LIN {X 0,Y 467.337,Z 283.456,A -85,B 0,C 180,E1 -7628.382,E2 -7628.382} C_VEL
LIN {X 0,Y 467.091,Z 291.095,A -85,B 0,C 180,E1 -7631.581,E2 -7631.581} C_VEL
LIN {X 0,Y 466.943,Z 298.315,A -85,B 0,C 180,E1 -7634.545,E2 -7634.545} C_VEL
LIN {X 0,Y 469.161,Z 311.668,A -85,B 0,C 180,E1 -7634.985,E2 -7634.985} C_VEL
LIN {X 0,Y 470.055,Z 319.78,A -85,B 0,C 180,E1 -7635.331,E2 -7635.331} C_VEL
LIN {X 0,Y 469.55,Z 331.872,A -85,B 0,C 180,E1 -7635.924,E2 -7635.924} C_VEL
LIN {X 0,Y 469.022,Z 343.532,A -85,B 0,C 180,E1 -7636.681,E2 -7636.681} C_VEL
LIN {X 0,Y 468.531,Z 353.937,A -85,B 0,C 180,E1 -7637.536,E2 -7637.536} C_VEL
LIN {X 0,Y 468.153,Z 363.71,A -85,B 0,C 180,E1 -7638.527,E2 -7638.527} C_VEL
LIN {X 0,Y 467.611,Z 372.508,A -85,B 0,C 180,E1 -7639.61,E2 -7639.61} C_VEL
LIN {X 0,Y 467.264,Z 381.091,A -85,B 0,C 180,E1 -7640.914,E2 -7640.914} C_VEL
LIN {X 0,Y 466.991,Z 387.971,A -85,B 0,C 180,E1 -7642.216,E2 -7642.216} C_VEL
LIN {X 0,Y 466.835,Z 393.494,A -85,B 0,C 180,E1 -7643.519,E2 -7643.519} C_VEL
LIN {X 0,Y 466.738,Z 397.815,A -85,B 0,C 180,E1 -7644.817,E2 -7644.817} C_VEL
LIN {X 0,Y 466.647,Z 400.107,A -85,B 0,C 180,E1 -7645.682,E2 -7645.682} C_VEL
LIN {X 0,Y 466.689,Z 401.966,A -85,B 0,C 180,E1 -7646.547,E2 -7646.547} C_VEL
LIN {X 0,Y 466.663,Z 403.358,A -85,B 0,C 180,E1 -7647.411,E2 -7647.411} C_VEL
LIN {X 0,Y 466.619,Z 404.96,A -85,B 0,C 180,E1 -7649.137,E2 -7649.137} C_VEL
LIN {X 0,Y 466.599,Z 405.172,A -85,B 0,C 180,E1 -7650,E2 -7650} C_VEL
LIN {X 0,Y 466.619,Z 404.953,A -85,B 0,C 180,E1 -7650.863,E2 -7650.863} C_VEL
LIN {X 0,Y 466.663,Z 403.347,A -85,B 0,C 180,E1 -7652.59,E2 -7652.59} C_VEL
LIN {X 0,Y 466.69,Z 401.945,A -85,B 0,C 180,E1 -7653.453,E2 -7653.453} C_VEL
LIN {X 0,Y 466.69,Z 399,A -85,B 0,C 180,E1 -7654.751,E2 -7654.751} C_VEL
LIN {X 0,Y 466.756,Z 395.011,A -85,B 0,C 180,E1 -7656.05,E2 -7656.05} C_VEL
LIN {X 0,Y 466.951,Z 388.871,A -85,B 0,C 180,E1 -7657.567,E2 -7657.567} C_VEL
LIN {X 0,Y 467.212,Z 382.165,A -85,B 0,C 180,E1 -7658.869,E2 -7658.869} C_VEL
LIN {X 0,Y 467.563,Z 373.843,A -85,B 0,C 180,E1 -7660.172,E2 -7660.172} C_VEL
LIN {X 0,Y 468.003,Z 365.294,A -85,B 0,C 180,E1 -7661.257,E2 -7661.257} C_VEL
LIN {X 0,Y 468.46,Z 355.172,A -85,B 0,C 180,E1 -7662.302,E2 -7662.302} C_VEL
LIN {X 0,Y 468.936,Z 344.257,A -85,B 0,C 180,E1 -7663.212,E2 -7663.212} C_VEL
LIN {X 0,Y 469.451,Z 332.748,A -85,B 0,C 180,E1 -7663.969,E2 -7663.969} C_VEL
LIN {X 0,Y 469.903,Z 320.822,A -85,B 0,C 180,E1 -7664.563,E2 -7664.563} C_VEL
LIN {X 0,Y 469.607,Z 315.894,A -85,B 0,C 180,E1 -7664.774,E2 -7664.774} C_VEL
LIN {X 0,Y 467.679,Z 303.276,A -85,B 0,C 180,E1 -7665.226,E2 -7665.226} C_VEL
LIN {X 0,Y 466.927,Z 298.392,A -85,B 0,C 180,E1 -7665.377,E2 -7665.377} C_VEL
LIN {X 0,Y 467.1,Z 290.512,A -85,B 0,C 180,E1 -7668.575,E2 -7668.575} C_VEL
LIN {X 0,Y 467.335,Z 283.121,A -85,B 0,C 180,E1 -7671.619,E2 -7671.619} C_VEL
LIN {X 0,Y 467.51,Z 275.327,A -85,B 0,C 180,E1 -7674.892,E2 -7674.892} C_VEL
LIN {X 0,Y 467.742,Z 268.646,A -85,B 0,C 180,E1 -7677.76,E2 -7677.76} C_VEL
LIN {X 0,Y 467.985,Z 261.965,A -85,B 0,C 180,E1 -7680.703,E2 -7680.703} C_VEL
LIN {X 0,Y 468.255,Z 256.383,A -85,B 0,C 180,E1 -7683.22,E2 -7683.22} C_VEL
LIN {X 0,Y 468.388,Z 250.837,A -85,B 0,C 180,E1 -7685.815,E2 -7685.815} C_VEL
LIN {X 0,Y 467.612,Z 245.311,A -85,B 0,C 180,E1 -7688.559,E2 -7688.559} C_VEL
LIN {X 0,Y 467.556,Z 245.245,A -85,B 0,C 180,E1 -7691.404,E2 -7691.404} C_VEL
LIN {X 0,Y 467.552,Z 245.247,A -85,B 0,C 180,E1 -7694.948,E2 -7694.948} C_VEL
LIN {X 0,Y 467.554,Z 245.247,A -85,B 0,C 180,E1 -7698.594,E2 -7698.594} C_VEL
LIN {X 0,Y 467.535,Z 245.244,A -85,B 0,C 180,E1 -7701.412,E2 -7701.412} C_VEL
LIN {X 0,Y 467.545,Z 245.247,A -85,B 0,C 180,E1 -7704.262,E2 -7704.262} C_VEL
LIN {X 0,Y 467.575,Z 245.24,A -85,B 0,C 180,E1 -7707.32,E2 -7707.32} C_VEL
LIN {X 0,Y 467.547,Z 245.245,A -85,B 0,C 180,E1 -7710.67,E2 -7710.67} C_VEL
LIN {X 0,Y 467.552,Z 245.243,A -85,B 0,C 180,E1 -7713.195,E2 -7713.195} C_VEL
LIN {X 0,Y 467.583,Z 245.24,A -85,B 0,C 180,E1 -7716.468,E2 -7716.468} C_VEL
LIN {X 0,Y 467.615,Z 245.238,A -85,B 0,C 180,E1 -7719.776,E2 -7719.776} C_VEL
LIN {X 0,Y 467.591,Z 245.239,A -85,B 0,C 180,E1 -7722.505,E2 -7722.505} C_VEL
LIN {X 0,Y 467.598,Z 245.239,A -85,B 0,C 180,E1 -7725.195,E2 -7725.195} C_VEL
LIN {X 0,Y 467.648,Z 245.233,A -85,B 0,C 180,E1 -7727.853,E2 -7727.853} C_VEL
LIN {X 0,Y 467.673,Z 245.231,A -85,B 0,C 180,E1 -7731.356,E2 -7731.356} C_VEL
LIN {X 0,Y 467.734,Z 245.221,A -85,B 0,C 180,E1 -7733.962,E2 -7733.962} C_VEL
LIN {X 0,Y 467.85,Z 245.208,A -85,B 0,C 180,E1 -7737.416,E2 -7737.416} C_VEL
LIN {X 0,Y 467.872,Z 245.204,A -85,B 0,C 180,E1 -7739.999,E2 -7739.999} C_VEL
LIN {X 0,Y 467.851,Z 245.208,A -85,B 0,C 180,E1 -7742.582,E2 -7742.582} C_VEL
LIN {X 0,Y 467.738,Z 245.222,A -85,B 0,C 180,E1 -7746.036,E2 -7746.036} C_VEL
LIN {X 0,Y 467.673,Z 245.23,A -85,B 0,C 180,E1 -7748.642,E2 -7748.642} C_VEL
LIN {X 0,Y 467.646,Z 245.235,A -85,B 0,C 180,E1 -7752.145,E2 -7752.145} C_VEL
LIN {X 0,Y 467.628,Z 245.236,A -85,B 0,C 180,E1 -7755.694,E2 -7755.694} C_VEL
LIN {X 0,Y 467.606,Z 245.237,A -85,B 0,C 180,E1 -7758.764,E2 -7758.764} C_VEL
LIN {X 0,Y 467.569,Z 245.242,A -85,B 0,C 180,E1 -7761.268,E2 -7761.268} C_VEL
LIN {X 0,Y 467.561,Z 245.244,A -85,B 0,C 180,E1 -7763.943,E2 -7763.943} C_VEL
LIN {X 0,Y 467.615,Z 245.235,A -85,B 0,C 180,E1 -7766.799,E2 -7766.799} C_VEL
LIN {X 0,Y 467.575,Z 245.242,A -85,B 0,C 180,E1 -7769.735,E2 -7769.735} C_VEL
LIN {X 0,Y 467.571,Z 245.241,A -85,B 0,C 180,E1 -7772.758,E2 -7772.758} C_VEL
LIN {X 0,Y 467.545,Z 245.243,A -85,B 0,C 180,E1 -7775.889,E2 -7775.889} C_VEL
LIN {X 0,Y 467.606,Z 245.241,A -85,B 0,C 180,E1 -7779.141,E2 -7779.141} C_VEL
LIN {X 0,Y 467.606,Z 245.237,A -85,B 0,C 180,E1 -7782.571,E2 -7782.571} C_VEL
LIN {X 0,Y 467.554,Z 245.241,A -85,B 0,C 180,E1 -7786.177,E2 -7786.177} C_VEL
LIN {X 0,Y 467.569,Z 245.246,A -85,B 0,C 180,E1 -7788.722,E2 -7788.722} C_VEL
LIN {X 0,Y 467.553,Z 245.242,A -85,B 0,C 180,E1 -7791.955,E2 -7791.955} C_VEL
LIN {X 0,Y 467.554,Z 245.242,A -85,B 0,C 180,E1 -7795.167,E2 -7795.167} C_VEL
LIN {X 0,Y 467.57,Z 245.245,A -85,B 0,C 180,E1 -7798.26,E2 -7798.26} C_VEL
LIN {X 0,Y 467.562,Z 245.241,A -85,B 0,C 180,E1 -7801.25,E2 -7801.25} C_VEL
LIN {X 0,Y 467.576,Z 245.245,A -85,B 0,C 180,E1 -7804.159,E2 -7804.159} C_VEL
LIN {X 0,Y 467.497,Z 245.249,A -85,B 0,C 180,E1 -7806.992,E2 -7806.992} C_VEL
LIN {X 0,Y 467.412,Z 245.264,A -85,B 0,C 180,E1 -7807.921,E2 -7807.921} C_VEL
LIN {X 0,Y 467.395,Z 246.234,A -85,B 0,C 180,E1 -7808.846,E2 -7808.846} C_VEL
LIN {X 0,Y 467.382,Z 250.183,A -85,B 0,C 180,E1 -7811.593,E2 -7811.593} C_VEL
LIN {X 0,Y 467.274,Z 254.14,A -85,B 0,C 180,E1 -7814.293,E2 -7814.293} C_VEL
LIN {X 0,Y 467.221,Z 255.612,A -85,B 0,C 180,E1 -7815.284,E2 -7815.284} C_VEL
LIN {X 0,Y 466.522,Z 256.725,A -85,B 0,C 180,E1 -7815.991,E2 -7815.991} C_VEL
LIN {X 0,Y 463.655,Z 258.714,A -85,B 0,C 180,E1 -7817.135,E2 -7817.135} C_VEL
LIN {X 0,Y 461.228,Z 260.326,A -85,B 0,C 180,E1 -7818.057,E2 -7818.057} C_VEL
LIN {X 0,Y 460.157,Z 261.495,A -85,B 0,C 180,E1 -7818.771,E2 -7818.771} C_VEL
LIN {X 0,Y 460.054,Z 261.867,A -85,B 0,C 180,E1 -7819.014,E2 -7819.014} C_VEL
LIN {X 0,Y 459.985,Z 266.526,A -85,B 0,C 180,E1 -7822.096,E2 -7822.096} C_VEL
LIN {X 0,Y 459.995,Z 269.228,A -85,B 0,C 180,E1 -7823.861,E2 -7823.861} C_VEL
LIN {X 0,Y 459.921,Z 273.289,A -85,B 0,C 180,E1 -7826.496,E2 -7826.496} C_VEL
LIN {X 0,Y 459.772,Z 275.027,A -85,B 0,C 180,E1 -7827.509,E2 -7827.509} C_VEL
LIN {X 0,Y 462.387,Z 288.038,A -85,B 0,C 180,E1 -7827.972,E2 -7827.972} C_VEL
LIN {X 0,Y 463.251,Z 293.332,A -85,B 0,C 180,E1 -7828.207,E2 -7828.207} C_VEL
LIN {X 0,Y 462.781,Z 305.595,A -85,B 0,C 180,E1 -7828.803,E2 -7828.803} C_VEL
LIN {X 0,Y 462.304,Z 317.382,A -85,B 0,C 180,E1 -7829.564,E2 -7829.564} C_VEL
LIN {X 0,Y 461.762,Z 329.095,A -85,B 0,C 180,E1 -7830.545,E2 -7830.545} C_VEL
LIN {X 0,Y 461.249,Z 338.561,A -85,B 0,C 180,E1 -7831.528,E2 -7831.528} C_VEL
LIN {X 0,Y 460.775,Z 347.211,A -85,B 0,C 180,E1 -7832.623,E2 -7832.623} C_VEL
LIN {X 0,Y 460.361,Z 355.626,A -85,B 0,C 180,E1 -7833.939,E2 -7833.939} C_VEL
LIN {X 0,Y 459.997,Z 362.401,A -85,B 0,C 180,E1 -7835.26,E2 -7835.26} C_VEL
LIN {X 0,Y 459.885,Z 367.999,A -85,B 0,C 180,E1 -7836.633,E2 -7836.633} C_VEL
LIN {X 0,Y 459.742,Z 372.063,A -85,B 0,C 180,E1 -7837.908,E2 -7837.908} C_VEL
LIN {X 0,Y 459.618,Z 374.329,A -85,B 0,C 180,E1 -7838.795,E2 -7838.795} C_VEL
LIN {X 0,Y 459.525,Z 376.121,A -85,B 0,C 180,E1 -7839.685,E2 -7839.685} C_VEL
LIN {X 0,Y 459.538,Z 377.468,A -85,B 0,C 180,E1 -7840.575,E2 -7840.575} C_VEL
LIN {X 0,Y 459.549,Z 378.692,A -85,B 0,C 180,E1 -7841.836,E2 -7841.836} C_VEL
LIN {X 0,Y 459.433,Z 379.083,A -85,B 0,C 180,E1 -7843.265,E2 -7843.265} C_VEL
LIN {X 0,Y 459.442,Z 378.784,A -85,B 0,C 180,E1 -7844.167,E2 -7844.167} C_VEL
LIN {X 0,Y 459.507,Z 377.557,A -85,B 0,C 180,E1 -7845.521,E2 -7845.521} C_VEL
LIN {X 0,Y 459.619,Z 374.388,A -85,B 0,C 180,E1 -7847.347,E2 -7847.347} C_VEL
LIN {X 0,Y 459.789,Z 370.739,A -85,B 0,C 180,E1 -7848.722,E2 -7848.722} C_VEL
LIN {X 0,Y 459.959,Z 365.869,A -85,B 0,C 180,E1 -7850.108,E2 -7850.108} C_VEL
LIN {X 0,Y 460.265,Z 359.619,A -85,B 0,C 180,E1 -7851.497,E2 -7851.497} C_VEL
LIN {X 0,Y 460.667,Z 351.74,A -85,B 0,C 180,E1 -7852.894,E2 -7852.894} C_VEL
LIN {X 0,Y 461.173,Z 342.78,A -85,B 0,C 180,E1 -7854.156,E2 -7854.156} C_VEL
LIN {X 0,Y 461.731,Z 332.286,A -85,B 0,C 180,E1 -7855.346,E2 -7855.346} C_VEL
LIN {X 0,Y 462.268,Z 321.584,A -85,B 0,C 180,E1 -7856.315,E2 -7856.315} C_VEL
LIN {X 0,Y 462.77,Z 310.611,A -85,B 0,C 180,E1 -7857.103,E2 -7857.103} C_VEL
LIN {X 0,Y 463.317,Z 299.025,A -85,B 0,C 180,E1 -7857.747,E2 -7857.747} C_VEL
LIN {X 0,Y 463.379,Z 292.5,A -85,B 0,C 180,E1 -7858.045,E2 -7858.045} C_VEL
LIN {X 0,Y 460.857,Z 279.894,A -85,B 0,C 180,E1 -7858.577,E2 -7858.577} C_VEL
LIN {X 0,Y 459.719,Z 275.001,A -85,B 0,C 180,E1 -7858.759,E2 -7858.759} C_VEL
LIN {X 0,Y 459.8,Z 271.128,A -85,B 0,C 180,E1 -7861.31,E2 -7861.31} C_VEL
LIN {X 0,Y 459.943,Z 266.479,A -85,B 0,C 180,E1 -7864.427,E2 -7864.427} C_VEL
LIN {X 0,Y 460.058,Z 261.784,A -85,B 0,C 180,E1 -7867.665,E2 -7867.665} C_VEL
LIN {X 0,Y 460.159,Z 258.147,A -85,B 0,C 180,E1 -7870.215,E2 -7870.215} C_VEL
LIN {X 0,Y 460.334,Z 253.735,A -85,B 0,C 180,E1 -7873.394,E2 -7873.394} C_VEL
LIN {X 0,Y 460.478,Z 250.436,A -85,B 0,C 180,E1 -7875.833,E2 -7875.833} C_VEL
LIN {X 0,Y 460.5,Z 247.076,A -85,B 0,C 180,E1 -7878.4,E2 -7878.4} C_VEL
LIN {X 0,Y 460.468,Z 246.334,A -85,B 0,C 180,E1 -7878.984,E2 -7878.984} C_VEL
LIN {X 0,Y 460.503,Z 246.128,A -85,B 0,C 180,E1 -7881.266,E2 -7881.266} C_VEL
LIN {X 0,Y 460.5,Z 246.126,A -85,B 0,C 180,E1 -7884.555,E2 -7884.555} C_VEL
LIN {X 0,Y 460.519,Z 246.123,A -85,B 0,C 180,E1 -7887.716,E2 -7887.716} C_VEL
LIN {X 0,Y 460.534,Z 246.119,A -85,B 0,C 180,E1 -7890.77,E2 -7890.77} C_VEL
LIN {X 0,Y 460.55,Z 246.118,A -85,B 0,C 180,E1 -7893.735,E2 -7893.735} C_VEL
LIN {X 0,Y 460.539,Z 246.118,A -85,B 0,C 180,E1 -7896.625,E2 -7896.625} C_VEL
LIN {X 0,Y 460.561,Z 246.117,A -85,B 0,C 180,E1 -7899.455,E2 -7899.455} C_VEL
LIN {X 0,Y 460.547,Z 246.118,A -85,B 0,C 180,E1 -7902.231,E2 -7902.231} C_VEL
LIN {X 0,Y 460.556,Z 246.116,A -85,B 0,C 180,E1 -7904.966,E2 -7904.966} C_VEL
LIN {X 0,Y 460.6,Z 246.113,A -85,B 0,C 180,E1 -7908.56,E2 -7908.56} C_VEL
LIN {X 0,Y 460.684,Z 246.099,A -85,B 0,C 180,E1 -7912.109,E2 -7912.109} C_VEL
LIN {X 0,Y 460.681,Z 246.102,A -85,B 0,C 180,E1 -7914.749,E2 -7914.749} C_VEL
LIN {X 0,Y 460.816,Z 246.087,A -85,B 0,C 180,E1 -7917.379,E2 -7917.379} C_VEL
LIN {X 0,Y 460.839,Z 246.08,A -85,B 0,C 180,E1 -7920.001,E2 -7920.001} C_VEL
LIN {X 0,Y 460.817,Z 246.083,A -85,B 0,C 180,E1 -7922.623,E2 -7922.623} C_VEL
LIN {X 0,Y 460.691,Z 246.099,A -85,B 0,C 180,E1 -7926.131,E2 -7926.131} C_VEL
LIN {X 0,Y 460.62,Z 246.108,A -85,B 0,C 180,E1 -7928.777,E2 -7928.777} C_VEL
LIN {X 0,Y 460.605,Z 246.113,A -85,B 0,C 180,E1 -7932.446,E2 -7932.446} C_VEL
LIN {X 0,Y 460.593,Z 246.114,A -85,B 0,C 180,E1 -7935.999,E2 -7935.999} C_VEL
LIN {X 0,Y 460.563,Z 246.118,A -85,B 0,C 180,E1 -7938.903,E2 -7938.903} C_VEL
LIN {X 0,Y 460.509,Z 246.126,A -85,B 0,C 180,E1 -7941.487,E2 -7941.487} C_VEL
LIN {X 0,Y 460.534,Z 246.123,A -85,B 0,C 180,E1 -7944.334,E2 -7944.334} C_VEL
LIN {X 0,Y 460.531,Z 246.123,A -85,B 0,C 180,E1 -7947.247,E2 -7947.247} C_VEL
LIN {X 0,Y 460.503,Z 246.125,A -85,B 0,C 180,E1 -7950.241,E2 -7950.241} C_VEL
LIN {X 0,Y 460.525,Z 246.122,A -85,B 0,C 180,E1 -7953.326,E2 -7953.326} C_VEL
LIN {X 0,Y 460.472,Z 246.129,A -85,B 0,C 180,E1 -7956.531,E2 -7956.531} C_VEL
LIN {X 0,Y 460.529,Z 246.119,A -85,B 0,C 180,E1 -7959.864,E2 -7959.864} C_VEL
LIN {X 0,Y 460.511,Z 246.124,A -85,B 0,C 180,E1 -7962.902,E2 -7962.902} C_VEL
LIN {X 0,Y 460.501,Z 246.126,A -85,B 0,C 180,E1 -7965.833,E2 -7965.833} C_VEL
LIN {X 0,Y 460.515,Z 246.126,A -85,B 0,C 180,E1 -7968.988,E2 -7968.988} C_VEL
LIN {X 0,Y 460.544,Z 246.294,A -85,B 0,C 180,E1 -7970.039,E2 -7970.039} C_VEL
LIN {X 0,Y 461.414,Z 251.524,A -85,B 0,C 180,E1 -7973.014,E2 -7973.014} C_VEL
LIN {X 0,Y 461.641,Z 255.871,A -85,B 0,C 180,E1 -7975.296,E2 -7975.296} C_VEL
LIN {X 0,Y 461.246,Z 262.522,A -85,B 0,C 180,E1 -7978.57,E2 -7978.57} C_VEL
LIN {X 0,Y 460.92,Z 268.312,A -85,B 0,C 180,E1 -7981.295,E2 -7981.295} C_VEL
LIN {X 0,Y 460.542,Z 275.812,A -85,B 0,C 180,E1 -7984.705,E2 -7984.705} C_VEL
LIN {X 0,Y 460.29,Z 283.369,A -85,B 0,C 180,E1 -7988.033,E2 -7988.033} C_VEL
LIN {X 0,Y 460.019,Z 291.021,A -85,B 0,C 180,E1 -7991.302,E2 -7991.302} C_VEL
LIN {X 0,Y 459.866,Z 298.093,A -85,B 0,C 180,E1 -7994.271,E2 -7994.271} C_VEL
LIN {X 0,Y 462.203,Z 311.72,A -85,B 0,C 180,E1 -7994.741,E2 -7994.741} C_VEL
LIN {X 0,Y 463.181,Z 320.041,A -85,B 0,C 180,E1 -7995.108,E2 -7995.108} C_VEL
LIN {X 0,Y 462.671,Z 332.016,A -85,B 0,C 180,E1 -7995.71,E2 -7995.71} C_VEL
LIN {X 0,Y 462.121,Z 343.569,A -85,B 0,C 180,E1 -7996.478,E2 -7996.478} C_VEL
LIN {X 0,Y 461.565,Z 354.304,A -85,B 0,C 180,E1 -7997.381,E2 -7997.381} C_VEL
LIN {X 0,Y 461.173,Z 363.657,A -85,B 0,C 180,E1 -7998.351,E2 -7998.351} C_VEL
LIN {X 0,Y 460.602,Z 372.425,A -85,B 0,C 180,E1 -7999.45,E2 -7999.45} C_VEL
LIN {X 0,Y 460.231,Z 380.975,A -85,B 0,C 180,E1 -8000.774,E2 -8000.774} C_VEL
LIN {X 0,Y 459.93,Z 387.835,A -85,B 0,C 180,E1 -8002.096,E2 -8002.096} C_VEL
LIN {X 0,Y 459.744,Z 393.784,A -85,B 0,C 180,E1 -8003.539,E2 -8003.539} C_VEL
LIN {X 0,Y 459.618,Z 398.866,A -85,B 0,C 180,E1 -8005.176,E2 -8005.176} C_VEL
LIN {X 0,Y 459.584,Z 401.786,A -85,B 0,C 180,E1 -8006.493,E2 -8006.493} C_VEL
LIN {X 0,Y 459.585,Z 403.173,A -85,B 0,C 180,E1 -8007.371,E2 -8007.371} C_VEL
LIN {X 0,Y 459.522,Z 404.766,A -85,B 0,C 180,E1 -8009.124,E2 -8009.124} C_VEL
LIN {X 0,Y 459.53,Z 404.972,A -85,B 0,C 180,E1 -8010,E2 -8010} C_VEL
LIN {X 0,Y 459.521,Z 404.133,A -85,B 0,C 180,E1 -8011.753,E2 -8011.753} C_VEL
LIN {X 0,Y 459.585,Z 403.133,A -85,B 0,C 180,E1 -8012.629,E2 -8012.629} C_VEL
LIN {X 0,Y 459.585,Z 401.722,A -85,B 0,C 180,E1 -8013.507,E2 -8013.507} C_VEL
LIN {X 0,Y 459.618,Z 398.769,A -85,B 0,C 180,E1 -8014.824,E2 -8014.824} C_VEL
LIN {X 0,Y 459.716,Z 393.725,A -85,B 0,C 180,E1 -8016.431,E2 -8016.431} C_VEL
LIN {X 0,Y 459.911,Z 387.593,A -85,B 0,C 180,E1 -8017.905,E2 -8017.905} C_VEL
LIN {X 0,Y 460.231,Z 380.642,A -85,B 0,C 180,E1 -8019.227,E2 -8019.227} C_VEL
LIN {X 0,Y 460.594,Z 371.921,A -85,B 0,C 180,E1 -8020.55,E2 -8020.55} C_VEL
LIN {X 0,Y 461.092,Z 362.99,A -85,B 0,C 180,E1 -8021.651,E2 -8021.651} C_VEL
LIN {X 0,Y 461.59,Z 352.085,A -85,B 0,C 180,E1 -8022.743,E2 -8022.743} C_VEL
LIN {X 0,Y 462.117,Z 340.786,A -85,B 0,C 180,E1 -8023.634,E2 -8023.634} C_VEL
LIN {X 0,Y 462.693,Z 328.254,A -85,B 0,C 180,E1 -8024.402,E2 -8024.402} C_VEL
LIN {X 0,Y 462.962,Z 318.886,A -85,B 0,C 180,E1 -8024.843,E2 -8024.843} C_VEL
LIN {X 0,Y 461.078,Z 305.955,A -85,B 0,C 180,E1 -8025.356,E2 -8025.356} C_VEL
LIN {X 0,Y 459.847,Z 298.205,A -85,B 0,C 180,E1 -8025.599,E2 -8025.599} C_VEL
LIN {X 0,Y 460.07,Z 289.556,A -85,B 0,C 180,E1 -8029.173,E2 -8029.173} C_VEL
LIN {X 0,Y 460.281,Z 281.788,A -85,B 0,C 180,E1 -8032.44,E2 -8032.44} C_VEL
LIN {X 0,Y 460.561,Z 273.953,A -85,B 0,C 180,E1 -8035.799,E2 -8035.799} C_VEL
LIN {X 0,Y 460.826,Z 266.206,A -85,B 0,C 180,E1 -8039.21,E2 -8039.21} C_VEL
LIN {X 0,Y 461.165,Z 259.53,A -85,B 0,C 180,E1 -8042.234,E2 -8042.234} C_VEL
LIN {X 0,Y 461.405,Z 252.861,A -85,B 0,C 180,E1 -8045.366,E2 -8045.366} C_VEL
LIN {X 0,Y 460.917,Z 248.389,A -85,B 0,C 180,E1 -8047.582,E2 -8047.582} C_VEL
LIN {X 0,Y 460.555,Z 246.12,A -85,B 0,C 180,E1 -8048.822,E2 -8048.822} C_VEL
LIN {X 0,Y 460.471,Z 246.126,A -85,B 0,C 180,E1 -8052.186,E2 -8052.186} C_VEL
LIN {X 0,Y 460.494,Z 246.122,A -85,B 0,C 180,E1 -8055.408,E2 -8055.408} C_VEL
LIN {X 0,Y 460.51,Z 246.122,A -85,B 0,C 180,E1 -8058.986,E2 -8058.986} C_VEL
LIN {X 0,Y 460.477,Z 246.127,A -85,B 0,C 180,E1 -8062.374,E2 -8062.374} C_VEL
LIN {X 0,Y 460.529,Z 246.118,A -85,B 0,C 180,E1 -8065.621,E2 -8065.621} C_VEL
LIN {X 0,Y 460.533,Z 246.118,A -85,B 0,C 180,E1 -8068.743,E2 -8068.743} C_VEL
LIN {X 0,Y 460.534,Z 246.122,A -85,B 0,C 180,E1 -8072.263,E2 -8072.263} C_VEL
LIN {X 0,Y 460.528,Z 246.118,A -85,B 0,C 180,E1 -8074.703,E2 -8074.703} C_VEL
LIN {X 0,Y 460.504,Z 246.123,A -85,B 0,C 180,E1 -8077.57,E2 -8077.57} C_VEL
LIN {X 0,Y 460.561,Z 246.115,A -85,B 0,C 180,E1 -8080.383,E2 -8080.383} C_VEL
LIN {X 0,Y 460.597,Z 246.111,A -85,B 0,C 180,E1 -8084.058,E2 -8084.058} C_VEL
LIN {X 0,Y 460.601,Z 246.113,A -85,B 0,C 180,E1 -8087.665,E2 -8087.665} C_VEL
LIN {X 0,Y 460.62,Z 246.109,A -85,B 0,C 180,E1 -8091.223,E2 -8091.223} C_VEL
LIN {X 0,Y 460.7,Z 246.098,A -85,B 0,C 180,E1 -8093.869,E2 -8093.869} C_VEL
LIN {X 0,Y 460.815,Z 246.085,A -85,B 0,C 180,E1 -8097.377,E2 -8097.377} C_VEL
LIN {X 0,Y 460.843,Z 246.08,A -85,B 0,C 180,E1 -8099.999,E2 -8099.999} C_VEL
LIN {X 0,Y 460.816,Z 246.084,A -85,B 0,C 180,E1 -8102.621,E2 -8102.621} C_VEL
LIN {X 0,Y 460.703,Z 246.1,A -85,B 0,C 180,E1 -8106.129,E2 -8106.129} C_VEL
LIN {X 0,Y 460.62,Z 246.108,A -85,B 0,C 180,E1 -8108.775,E2 -8108.775} C_VEL
LIN {X 0,Y 460.602,Z 246.11,A -85,B 0,C 180,E1 -8112.444,E2 -8112.444} C_VEL
LIN {X 0,Y 460.589,Z 246.114,A -85,B 0,C 180,E1 -8115.997,E2 -8115.997} C_VEL
LIN {X 0,Y 460.559,Z 246.114,A -85,B 0,C 180,E1 -8118.901,E2 -8118.901} C_VEL
LIN {X 0,Y 460.504,Z 246.124,A -85,B 0,C 180,E1 -8121.485,E2 -8121.485} C_VEL
LIN {X 0,Y 460.53,Z 246.118,A -85,B 0,C 180,E1 -8124.332,E2 -8124.332} C_VEL
LIN {X 0,Y 460.572,Z 246.115,A -85,B 0,C 180,E1 -8127.242,E2 -8127.242} C_VEL
LIN {X 0,Y 460.515,Z 246.119,A -85,B 0,C 180,E1 -8130.238,E2 -8130.238} C_VEL
LIN {X 0,Y 460.517,Z 246.124,A -85,B 0,C 180,E1 -8133.324,E2 -8133.324} C_VEL
LIN {X 0,Y 460.468,Z 246.125,A -85,B 0,C 180,E1 -8136.528,E2 -8136.528} C_VEL
LIN {X 0,Y 460.566,Z 246.112,A -85,B 0,C 180,E1 -8139.857,E2 -8139.857} C_VEL
LIN {X 0,Y 460.53,Z 246.123,A -85,B 0,C 180,E1 -8142.904,E2 -8142.904} C_VEL
LIN {X 0,Y 460.506,Z 246.118,A -85,B 0,C 180,E1 -8145.829,E2 -8145.829} C_VEL
LIN {X 0,Y 460.521,Z 246.121,A -85,B 0,C 180,E1 -8148.989,E2 -8148.989} C_VEL
LIN {X 0,Y 460.513,Z 246.119,A -85,B 0,C 180,E1 -8151.267,E2 -8151.267} C_VEL
LIN {X 0,Y 460.5,Z 246.126,A -85,B 0,C 180,E1 -8154.554,E2 -8154.554} C_VEL
LIN {X 0,Y 460.519,Z 246.119,A -85,B 0,C 180,E1 -8157.715,E2 -8157.715} C_VEL
LIN {X 0,Y 460.526,Z 246.119,A -85,B 0,C 180,E1 -8160.769,E2 -8160.769} C_VEL
LIN {X 0,Y 460.53,Z 246.119,A -85,B 0,C 180,E1 -8163.733,E2 -8163.733} C_VEL
LIN {X 0,Y 460.493,Z 246.123,A -85,B 0,C 180,E1 -8166.622,E2 -8166.622} C_VEL
LIN {X 0,Y 460.394,Z 246.136,A -85,B 0,C 180,E1 -8167.566,E2 -8167.566} C_VEL
LIN {X 0,Y 460.351,Z 246.764,A -85,B 0,C 180,E1 -8168.628,E2 -8168.628} C_VEL
LIN {X 0,Y 460.336,Z 250.56,A -85,B 0,C 180,E1 -8171.301,E2 -8171.301} C_VEL
LIN {X 0,Y 460.208,Z 254.705,A -85,B 0,C 180,E1 -8174.168,E2 -8174.168} C_VEL
LIN {X 0,Y 460.179,Z 260.044,A -85,B 0,C 180,E1 -8177.796,E2 -8177.796} C_VEL
LIN {X 0,Y 460.054,Z 261.867,A -85,B 0,C 180,E1 -8179.014,E2 -8179.014} C_VEL
LIN {X 0,Y 459.332,Z 263.009,A -85,B 0,C 180,E1 -8179.73,E2 -8179.73} C_VEL
LIN {X 0,Y 456.425,Z 265.021,A -85,B 0,C 180,E1 -8180.889,E2 -8180.889} C_VEL
LIN {X 0,Y 454.015,Z 266.644,A -85,B 0,C 180,E1 -8181.824,E2 -8181.824} C_VEL
LIN {X 0,Y 453.012,Z 267.825,A -85,B 0,C 180,E1 -8182.548,E2 -8182.548} C_VEL
LIN {X 0,Y 452.946,Z 268.201,A -85,B 0,C 180,E1 -8182.793,E2 -8182.793} C_VEL
LIN {X 0,Y 452.9,Z 272.381,A -85,B 0,C 180,E1 -8185.55,E2 -8185.55} C_VEL
LIN {X 0,Y 452.753,Z 275.057,A -85,B 0,C 180,E1 -8187.275,E2 -8187.275} C_VEL
LIN {X 0,Y 455.252,Z 288.015,A -85,B 0,C 180,E1 -8187.747,E2 -8187.747} C_VEL
LIN {X 0,Y 456.35,Z 293.838,A -85,B 0,C 180,E1 -8188.014,E2 -8188.014} C_VEL
LIN {X 0,Y 455.884,Z 305.059,A -85,B 0,C 180,E1 -8188.565,E2 -8188.565} C_VEL
LIN {X 0,Y 455.405,Z 317.014,A -85,B 0,C 180,E1 -8189.337,E2 -8189.337} C_VEL
LIN {X 0,Y 454.855,Z 327.71,A -85,B 0,C 180,E1 -8190.221,E2 -8190.221} C_VEL
LIN {X 0,Y 454.265,Z 338.411,A -85,B 0,C 180,E1 -8191.33,E2 -8191.33} C_VEL
LIN {X 0,Y 453.783,Z 347.119,A -85,B 0,C 180,E1 -8192.441,E2 -8192.441} C_VEL
LIN {X 0,Y 453.316,Z 355.609,A -85,B 0,C 180,E1 -8193.778,E2 -8193.778} C_VEL
LIN {X 0,Y 452.944,Z 362.424,A -85,B 0,C 180,E1 -8195.118,E2 -8195.118} C_VEL
LIN {X 0,Y 452.804,Z 368.465,A -85,B 0,C 180,E1 -8196.626,E2 -8196.626} C_VEL
LIN {X 0,Y 452.647,Z 372.78,A -85,B 0,C 180,E1 -8198.032,E2 -8198.032} C_VEL
LIN {X 0,Y 452.51,Z 374.934,A -85,B 0,C 180,E1 -8198.935,E2 -8198.935} C_VEL
LIN {X 0,Y 452.429,Z 376.625,A -85,B 0,C 180,E1 -8199.838,E2 -8199.838} C_VEL
LIN {X 0,Y 452.437,Z 377.905,A -85,B 0,C 180,E1 -8200.743,E2 -8200.743} C_VEL
LIN {X 0,Y 452.447,Z 378.918,A -85,B 0,C 180,E1 -8201.883,E2 -8201.883} C_VEL
LIN {X 0,Y 452.345,Z 379.25,A -85,B 0,C 180,E1 -8203.476,E2 -8203.476} C_VEL
LIN {X 0,Y 452.354,Z 378.883,A -85,B 0,C 180,E1 -8204.393,E2 -8204.393} C_VEL
LIN {X 0,Y 452.427,Z 377.709,A -85,B 0,C 180,E1 -8205.618,E2 -8205.618} C_VEL
LIN {X 0,Y 452.496,Z 375.156,A -85,B 0,C 180,E1 -8207.163,E2 -8207.163} C_VEL
LIN {X 0,Y 452.707,Z 371.21,A -85,B 0,C 180,E1 -8208.745,E2 -8208.745} C_VEL
LIN {X 0,Y 452.864,Z 367.133,A -85,B 0,C 180,E1 -8209.963,E2 -8209.963} C_VEL
LIN {X 0,Y 453.203,Z 360.564,A -85,B 0,C 180,E1 -8211.5,E2 -8211.5} C_VEL
LIN {X 0,Y 453.593,Z 353.619,A -85,B 0,C 180,E1 -8212.789,E2 -8212.789} C_VEL
LIN {X 0,Y 454.092,Z 345.186,A -85,B 0,C 180,E1 -8214.06,E2 -8214.06} C_VEL
LIN {X 0,Y 454.618,Z 336.264,A -85,B 0,C 180,E1 -8215.158,E2 -8215.158} C_VEL
LIN {X 0,Y 455.213,Z 325.906,A -85,B 0,C 180,E1 -8216.188,E2 -8216.188} C_VEL
LIN {X 0,Y 455.762,Z 314.997,A -85,B 0,C 180,E1 -8217.058,E2 -8217.058} C_VEL
LIN {X 0,Y 456.342,Z 303.508,A -85,B 0,C 180,E1 -8217.776,E2 -8217.776} C_VEL
LIN {X 0,Y 456.504,Z 293.308,A -85,B 0,C 180,E1 -8218.275,E2 -8218.275} C_VEL
LIN {X 0,Y 454.092,Z 281.17,A -85,B 0,C 180,E1 -8218.812,E2 -8218.812} C_VEL
LIN {X 0,Y 452.648,Z 275.183,A -85,B 0,C 180,E1 -8219.057,E2 -8219.057} C_VEL
LIN {X 0,Y 452.738,Z 270.993,A -85,B 0,C 180,E1 -8221.856,E2 -8221.856} C_VEL
LIN {X 0,Y 452.877,Z 266.334,A -85,B 0,C 180,E1 -8225.042,E2 -8225.042} C_VEL
LIN {X 0,Y 453.033,Z 261.603,A -85,B 0,C 180,E1 -8228.354,E2 -8228.354} C_VEL
LIN {X 0,Y 453.154,Z 256.782,A -85,B 0,C 180,E1 -8231.826,E2 -8231.826} C_VEL
LIN {X 0,Y 453.373,Z 253.147,A -85,B 0,C 180,E1 -8234.517,E2 -8234.517} C_VEL
LIN {X 0,Y 453.468,Z 249.862,A -85,B 0,C 180,E1 -8237.008,E2 -8237.008} C_VEL
LIN {X 0,Y 453.453,Z 247.009,A -85,B 0,C 180,E1 -8239.414,E2 -8239.414} C_VEL
LIN {X 0,Y 453.458,Z 247.003,A -85,B 0,C 180,E1 -8242.813,E2 -8242.813} C_VEL
LIN {X 0,Y 453.465,Z 247.004,A -85,B 0,C 180,E1 -8246.088,E2 -8246.088} C_VEL
LIN {X 0,Y 453.47,Z 247,A -85,B 0,C 180,E1 -8249.242,E2 -8249.242} C_VEL
LIN {X 0,Y 453.524,Z 246.992,A -85,B 0,C 180,E1 -8252.298,E2 -8252.298} C_VEL
LIN {X 0,Y 453.503,Z 246.995,A -85,B 0,C 180,E1 -8255.266,E2 -8255.266} C_VEL
LIN {X 0,Y 453.524,Z 246.992,A -85,B 0,C 180,E1 -8258.398,E2 -8258.398} C_VEL
LIN {X 0,Y 453.51,Z 246.996,A -85,B 0,C 180,E1 -8261.009,E2 -8261.009} C_VEL
LIN {X 0,Y 453.564,Z 246.991,A -85,B 0,C 180,E1 -8263.877,E2 -8263.877} C_VEL
LIN {X 0,Y 453.552,Z 246.988,A -85,B 0,C 180,E1 -8267.472,E2 -8267.472} C_VEL
LIN {X 0,Y 453.582,Z 246.986,A -85,B 0,C 180,E1 -8271.088,E2 -8271.088} C_VEL
LIN {X 0,Y 453.655,Z 246.974,A -85,B 0,C 180,E1 -8273.776,E2 -8273.776} C_VEL
LIN {X 0,Y 453.757,Z 246.966,A -85,B 0,C 180,E1 -8277.338,E2 -8277.338} C_VEL
LIN {X 0,Y 453.81,Z 246.955,A -85,B 0,C 180,E1 -8280.001,E2 -8280.001} C_VEL
LIN {X 0,Y 453.757,Z 246.963,A -85,B 0,C 180,E1 -8282.664,E2 -8282.664} C_VEL
LIN {X 0,Y 453.659,Z 246.975,A -85,B 0,C 180,E1 -8286.227,E2 -8286.227} C_VEL
LIN {X 0,Y 453.584,Z 246.984,A -85,B 0,C 180,E1 -8288.915,E2 -8288.915} C_VEL
LIN {X 0,Y 453.556,Z 246.992,A -85,B 0,C 180,E1 -8292.53,E2 -8292.53} C_VEL
LIN {X 0,Y 453.537,Z 246.992,A -85,B 0,C 180,E1 -8296.197,E2 -8296.197} C_VEL
LIN {X 0,Y 453.513,Z 246.996,A -85,B 0,C 180,E1 -8299.042,E2 -8299.042} C_VEL
LIN {X 0,Y 453.47,Z 247.003,A -85,B 0,C 180,E1 -8301.837,E2 -8301.837} C_VEL
LIN {X 0,Y 453.503,Z 247.001,A -85,B 0,C 180,E1 -8304.736,E2 -8304.736} C_VEL
LIN {X 0,Y 453.5,Z 246.999,A -85,B 0,C 180,E1 -8307.954,E2 -8307.954} C_VEL
LIN {X 0,Y 453.47,Z 247.003,A -85,B 0,C 180,E1 -8310.761,E2 -8310.761} C_VEL
LIN {X 0,Y 453.472,Z 247.001,A -85,B 0,C 180,E1 -8313.914,E2 -8313.914} C_VEL
LIN {X 0,Y 453.448,Z 247.002,A -85,B 0,C 180,E1 -8317.191,E2 -8317.191} C_VEL
LIN {X 0,Y 453.502,Z 246.996,A -85,B 0,C 180,E1 -8319.449,E2 -8319.449} C_VEL
LIN {X 0,Y 453.461,Z 247.003,A -85,B 0,C 180,E1 -8322.996,E2 -8322.996} C_VEL
LIN {X 0,Y 453.456,Z 247.002,A -85,B 0,C 180,E1 -8325.779,E2 -8325.779} C_VEL
LIN {X 0,Y 453.496,Z 246.999,A -85,B 0,C 180,E1 -8329.596,E2 -8329.596} C_VEL
LIN {X 0,Y 454.425,Z 252.628,A -85,B 0,C 180,E1 -8332.904,E2 -8332.904} C_VEL
LIN {X 0,Y 454.638,Z 256.744,A -85,B 0,C 180,E1 -8335.114,E2 -8335.114} C_VEL
LIN {X 0,Y 454.328,Z 261.957,A -85,B 0,C 180,E1 -8337.746,E2 -8337.746} C_VEL
LIN {X 0,Y 453.961,Z 268.284,A -85,B 0,C 180,E1 -8340.813,E2 -8340.813} C_VEL
LIN {X 0,Y 453.533,Z 275.748,A -85,B 0,C 180,E1 -8344.286,E2 -8344.286} C_VEL
LIN {X 0,Y 453.251,Z 283.29,A -85,B 0,C 180,E1 -8347.674,E2 -8347.674} C_VEL
LIN {X 0,Y 453.041,Z 289.788,A -85,B 0,C 180,E1 -8350.517,E2 -8350.517} C_VEL
LIN {X 0,Y 452.832,Z 297.904,A -85,B 0,C 180,E1 -8353.997,E2 -8353.997} C_VEL
LIN {X 0,Y 455.216,Z 311.642,A -85,B 0,C 180,E1 -8354.48,E2 -8354.48} C_VEL
LIN {X 0,Y 456.324,Z 321.665,A -85,B 0,C 180,E1 -8354.936,E2 -8354.936} C_VEL
LIN {X 0,Y 455.713,Z 333.987,A -85,B 0,C 180,E1 -8355.601,E2 -8355.601} C_VEL
LIN {X 0,Y 455.048,Z 346.499,A -85,B 0,C 180,E1 -8356.491,E2 -8356.491} C_VEL
LIN {X 0,Y 454.553,Z 356.142,A -85,B 0,C 180,E1 -8357.359,E2 -8357.359} C_VEL
LIN {X 0,Y 454.113,Z 365.546,A -85,B 0,C 180,E1 -8358.394,E2 -8358.394} C_VEL
LIN {X 0,Y 453.509,Z 373.915,A -85,B 0,C 180,E1 -8359.509,E2 -8359.509} C_VEL
LIN {X 0,Y 453.117,Z 382.114,A -85,B 0,C 180,E1 -8360.853,E2 -8360.853} C_VEL
LIN {X 0,Y 452.865,Z 387.717,A -85,B 0,C 180,E1 -8361.971,E2 -8361.971} C_VEL
LIN {X 0,Y 452.653,Z 394.09,A -85,B 0,C 180,E1 -8363.56,E2 -8363.56} C_VEL
LIN {X 0,Y 452.546,Z 398.706,A -85,B 0,C 180,E1 -8365.1,E2 -8365.1} C_VEL
LIN {X 0,Y 452.48,Z 401.613,A -85,B 0,C 180,E1 -8366.438,E2 -8366.438} C_VEL
LIN {X 0,Y 452.509,Z 402.993,A -85,B 0,C 180,E1 -8367.33,E2 -8367.33} C_VEL
LIN {X 0,Y 452.429,Z 404.574,A -85,B 0,C 180,E1 -8369.11,E2 -8369.11} C_VEL
LIN {X 0,Y 452.435,Z 404.771,A -85,B 0,C 180,E1 -8370,E2 -8370} C_VEL
LIN {X 0,Y 452.437,Z 403.919,A -85,B 0,C 180,E1 -8371.78,E2 -8371.78} C_VEL
LIN {X 0,Y 452.509,Z 402.913,A -85,B 0,C 180,E1 -8372.671,E2 -8372.671} C_VEL
LIN {X 0,Y 452.481,Z 401.491,A -85,B 0,C 180,E1 -8373.562,E2 -8373.562} C_VEL
LIN {X 0,Y 452.546,Z 398.527,A -85,B 0,C 180,E1 -8374.9,E2 -8374.9} C_VEL
LIN {X 0,Y 452.613,Z 393.956,A -85,B 0,C 180,E1 -8376.396,E2 -8376.396} C_VEL
LIN {X 0,Y 452.857,Z 387.312,A -85,B 0,C 180,E1 -8378.029,E2 -8378.029} C_VEL
LIN {X 0,Y 453.2,Z 380.335,A -85,B 0,C 180,E1 -8379.371,E2 -8379.371} C_VEL
LIN {X 0,Y 453.572,Z 371.578,A -85,B 0,C 180,E1 -8380.716,E2 -8380.716} C_VEL
LIN {X 0,Y 454.103,Z 362.613,A -85,B 0,C 180,E1 -8381.833,E2 -8381.833} C_VEL
LIN {X 0,Y 454.602,Z 352.363,A -85,B 0,C 180,E1 -8382.877,E2 -8382.877} C_VEL
LIN {X 0,Y 455.098,Z 341.877,A -85,B 0,C 180,E1 -8383.735,E2 -8383.735} C_VEL
LIN {X 0,Y 455.685,Z 329.667,A -85,B 0,C 180,E1 -8384.514,E2 -8384.514} C_VEL
LIN {X 0,Y 456,Z 319.48,A -85,B 0,C 180,E1 -8385.017,E2 -8385.017} C_VEL
LIN {X 0,Y 454.078,Z 306.106,A -85,B 0,C 180,E1 -8385.564,E2 -8385.564} C_VEL
LIN {X 0,Y 452.771,Z 298.065,A -85,B 0,C 180,E1 -8385.804,E2 -8385.804} C_VEL
LIN {X 0,Y 452.979,Z 290.425,A -85,B 0,C 180,E1 -8389.015,E2 -8389.015} C_VEL
LIN {X 0,Y 453.215,Z 282.67,A -85,B 0,C 180,E1 -8392.328,E2 -8392.328} C_VEL
LIN {X 0,Y 453.489,Z 274.894,A -85,B 0,C 180,E1 -8395.717,E2 -8395.717} C_VEL
LIN {X 0,Y 453.789,Z 267.107,A -85,B 0,C 180,E1 -8399.199,E2 -8399.199} C_VEL
LIN {X 0,Y 454.145,Z 260.433,A -85,B 0,C 180,E1 -8402.268,E2 -8402.268} C_VEL
LIN {X 0,Y 454.384,Z 253.76,A -85,B 0,C 180,E1 -8405.45,E2 -8405.45} C_VEL
LIN {X 0,Y 453.845,Z 249.054,A -85,B 0,C 180,E1 -8407.836,E2 -8407.836} C_VEL
LIN {X 0,Y 453.521,Z 246.996,A -85,B 0,C 180,E1 -8408.955,E2 -8408.955} C_VEL
LIN {X 0,Y 453.433,Z 247.002,A -85,B 0,C 180,E1 -8411.928,E2 -8411.928} C_VEL
LIN {X 0,Y 453.464,Z 246.997,A -85,B 0,C 180,E1 -8415.472,E2 -8415.472} C_VEL
LIN {X 0,Y 453.438,Z 247.001,A -85,B 0,C 180,E1 -8418.204,E2 -8418.204} C_VEL
LIN {X 0,Y 453.433,Z 247.005,A -85,B 0,C 180,E1 -8420.801,E2 -8420.801} C_VEL
LIN {X 0,Y 453.436,Z 247.002,A -85,B 0,C 180,E1 -8423.915,E2 -8423.915} C_VEL
LIN {X 0,Y 453.474,Z 246.997,A -85,B 0,C 180,E1 -8427.15,E2 -8427.15} C_VEL
LIN {X 0,Y 453.459,Z 247.003,A -85,B 0,C 180,E1 -8430.266,E2 -8430.266} C_VEL
LIN {X 0,Y 453.455,Z 247,A -85,B 0,C 180,E1 -8433.29,E2 -8433.29} C_VEL
LIN {X 0,Y 453.488,Z 246.998,A -85,B 0,C 180,E1 -8436.237,E2 -8436.237} C_VEL
LIN {X 0,Y 453.476,Z 246.998,A -85,B 0,C 180,E1 -8439.116,E2 -8439.116} C_VEL
LIN {X 0,Y 453.497,Z 246.998,A -85,B 0,C 180,E1 -8441.943,E2 -8441.943} C_VEL
LIN {X 0,Y 453.532,Z 246.991,A -85,B 0,C 180,E1 -8444.725,E2 -8444.725} C_VEL
LIN {X 0,Y 453.551,Z 246.988,A -85,B 0,C 180,E1 -8448.378,E2 -8448.378} C_VEL
LIN {X 0,Y 453.644,Z 246.977,A -85,B 0,C 180,E1 -8451.984,E2 -8451.984} C_VEL
LIN {X 0,Y 453.661,Z 246.976,A -85,B 0,C 180,E1 -8454.666,E2 -8454.666} C_VEL
LIN {X 0,Y 453.755,Z 246.965,A -85,B 0,C 180,E1 -8457.336,E2 -8457.336} C_VEL
LIN {X 0,Y 453.814,Z 246.956,A -85,B 0,C 180,E1 -8459.999,E2 -8459.999} C_VEL
LIN {X 0,Y 453.756,Z 246.963,A -85,B 0,C 180,E1 -8462.662,E2 -8462.662} C_VEL
LIN {X 0,Y 453.67,Z 246.976,A -85,B 0,C 180,E1 -8466.224,E2 -8466.224} C_VEL
LIN {X 0,Y 453.583,Z 246.985,A -85,B 0,C 180,E1 -8468.912,E2 -8468.912} C_VEL
LIN {X 0,Y 453.553,Z 246.988,A -85,B 0,C 180,E1 -8472.528,E2 -8472.528} C_VEL
LIN {X 0,Y 453.534,Z 246.991,A -85,B 0,C 180,E1 -8476.195,E2 -8476.195} C_VEL
LIN {X 0,Y 453.509,Z 246.993,A -85,B 0,C 180,E1 -8479.04,E2 -8479.04} C_VEL
LIN {X 0,Y 453.465,Z 247.001,A -85,B 0,C 180,E1 -8481.835,E2 -8481.835} C_VEL
LIN {X 0,Y 453.502,Z 246.993,A -85,B 0,C 180,E1 -8484.734,E2 -8484.734} C_VEL
LIN {X 0,Y 453.527,Z 246.991,A -85,B 0,C 180,E1 -8487.961,E2 -8487.961} C_VEL
LIN {X 0,Y 453.471,Z 246.997,A -85,B 0,C 180,E1 -8490.758,E2 -8490.758} C_VEL
LIN {X 0,Y 453.465,Z 246.997,A -85,B 0,C 180,E1 -8493.912,E2 -8493.912} C_VEL
LIN {X 0,Y 453.46,Z 247.003,A -85,B 0,C 180,E1 -8497.187,E2 -8497.187} C_VEL
LIN {X 0,Y 453.521,Z 246.991,A -85,B 0,C 180,E1 -8499.445,E2 -8499.445} C_VEL
LIN {X 0,Y 453.48,Z 247,A -85,B 0,C 180,E1 -8502.991,E2 -8502.991} C_VEL
LIN {X 0,Y 453.46,Z 246.996,A -85,B 0,C 180,E1 -8505.78,E2 -8505.78} C_VEL
LIN {X 0,Y 453.469,Z 246.997,A -85,B 0,C 180,E1 -8508.209,E2 -8508.209} C_VEL
LIN {X 0,Y 453.497,Z 246.997,A -85,B 0,C 180,E1 -8510.791,E2 -8510.791} C_VEL
LIN {X 0,Y 453.443,Z 247,A -85,B 0,C 180,E1 -8513.917,E2 -8513.917} C_VEL
LIN {X 0,Y 453.47,Z 246.996,A -85,B 0,C 180,E1 -8517.151,E2 -8517.151} C_VEL
LIN {X 0,Y 453.462,Z 247.003,A -85,B 0,C 180,E1 -8520.268,E2 -8520.268} C_VEL
LIN {X 0,Y 453.476,Z 246.996,A -85,B 0,C 180,E1 -8523.293,E2 -8523.293} C_VEL
LIN {X 0,Y 453.463,Z 247.002,A -85,B 0,C 180,E1 -8526.237,E2 -8526.237} C_VEL
LIN {X 0,Y 453.288,Z 247.025,A -85,B 0,C 180,E1 -8528.155,E2 -8528.155} C_VEL
LIN {X 0,Y 453.285,Z 250.994,A -85,B 0,C 180,E1 -8531.041,E2 -8531.041} C_VEL
LIN {X 0,Y 453.138,Z 256.245,A -85,B 0,C 180,E1 -8534.713,E2 -8534.713} C_VEL
LIN {X 0,Y 453.056,Z 261.578,A -85,B 0,C 180,E1 -8538.366,E2 -8538.366} C_VEL
LIN {X 0,Y 452.936,Z 266.963,A -85,B 0,C 180,E1 -8541.973,E2 -8541.973} C_VEL
LIN {X 0,Y 452.946,Z 268.201,A -85,B 0,C 180,E1 -8542.793,E2 -8542.793} C_VEL
LIN {X 0,Y 452.311,Z 269.358,A -85,B 0,C 180,E1 -8543.52,E2 -8543.52} C_VEL
LIN {X 0,Y 449.423,Z 271.382,A -85,B 0,C 180,E1 -8544.697,E2 -8544.697} C_VEL
LIN {X 0,Y 446.942,Z 273.016,A -85,B 0,C 180,E1 -8545.646,E2 -8545.646} C_VEL
LIN {X 0,Y 445.856,Z 274.213,A -85,B 0,C 180,E1 -8546.381,E2 -8546.381} C_VEL
LIN {X 0,Y 445.76,Z 274.598,A -85,B 0,C 180,E1 -8546.631,E2 -8546.631} C_VEL
LIN {X 0,Y 445.719,Z 275.447,A -85,B 0,C 180,E1 -8547.063,E2 -8547.063} C_VEL
LIN {X 0,Y 448.063,Z 287.578,A -85,B 0,C 180,E1 -8547.5,E2 -8547.5} C_VEL
LIN {X 0,Y 449.391,Z 295.57,A -85,B 0,C 180,E1 -8547.871,E2 -8547.871} C_VEL
LIN {X 0,Y 448.942,Z 306.422,A -85,B 0,C 180,E1 -8548.43,E2 -8548.43} C_VEL
LIN {X 0,Y 448.433,Z 318.099,A -85,B 0,C 180,E1 -8549.214,E2 -8549.214} C_VEL
LIN {X 0,Y 447.796,Z 329.774,A -85,B 0,C 180,E1 -8550.225,E2 -8550.225} C_VEL
LIN {X 0,Y 447.2,Z 340.161,A -85,B 0,C 180,E1 -8551.351,E2 -8551.351} C_VEL
LIN {X 0,Y 446.687,Z 348.581,A -85,B 0,C 180,E1 -8552.48,E2 -8552.48} C_VEL
LIN {X 0,Y 446.244,Z 356.795,A -85,B 0,C 180,E1 -8553.838,E2 -8553.838} C_VEL
LIN {X 0,Y 445.904,Z 362.43,A -85,B 0,C 180,E1 -8554.973,E2 -8554.973} C_VEL
LIN {X 0,Y 445.755,Z 367.916,A -85,B 0,C 180,E1 -8556.336,E2 -8556.336} C_VEL
LIN {X 0,Y 445.593,Z 372.237,A -85,B 0,C 180,E1 -8557.704,E2 -8557.704} C_VEL
LIN {X 0,Y 445.417,Z 375.5,A -85,B 0,C 180,E1 -8559.078,E2 -8559.078} C_VEL
LIN {X 0,Y 445.341,Z 377.122,A -85,B 0,C 180,E1 -8559.997,E2 -8559.997} C_VEL
LIN {X 0,Y 445.336,Z 378.333,A -85,B 0,C 180,E1 -8560.916,E2 -8560.916} C_VEL
LIN {X 0,Y 445.361,Z 379.147,A -85,B 0,C 180,E1 -8561.941,E2 -8561.941} C_VEL
LIN {X 0,Y 445.257,Z 379.418,A -85,B 0,C 180,E1 -8563.695,E2 -8563.695} C_VEL
LIN {X 0,Y 445.28,Z 378.966,A -85,B 0,C 180,E1 -8564.627,E2 -8564.627} C_VEL
LIN {X 0,Y 445.353,Z 377.862,A -85,B 0,C 180,E1 -8565.72,E2 -8565.72} C_VEL
LIN {X 0,Y 445.449,Z 374.978,A -85,B 0,C 180,E1 -8567.443,E2 -8567.443} C_VEL
LIN {X 0,Y 445.654,Z 371.337,A -85,B 0,C 180,E1 -8568.884,E2 -8568.884} C_VEL
LIN {X 0,Y 445.869,Z 366.615,A -85,B 0,C 180,E1 -8570.29,E2 -8570.29} C_VEL
LIN {X 0,Y 446.285,Z 359.671,A -85,B 0,C 180,E1 -8571.883,E2 -8571.883} C_VEL
LIN {X 0,Y 446.67,Z 352.676,A -85,B 0,C 180,E1 -8573.163,E2 -8573.163} C_VEL
LIN {X 0,Y 447.193,Z 344.617,A -85,B 0,C 180,E1 -8574.368,E2 -8574.368} C_VEL
LIN {X 0,Y 447.761,Z 334.684,A -85,B 0,C 180,E1 -8575.571,E2 -8575.571} C_VEL
LIN {X 0,Y 448.452,Z 323.955,A -85,B 0,C 180,E1 -8576.612,E2 -8576.612} C_VEL
LIN {X 0,Y 449.05,Z 312.508,A -85,B 0,C 180,E1 -8577.496,E2 -8577.496} C_VEL
LIN {X 0,Y 449.695,Z 300.577,A -85,B 0,C 180,E1 -8578.198,E2 -8578.198} C_VEL
LIN {X 0,Y 449.607,Z 293.749,A -85,B 0,C 180,E1 -8578.533,E2 -8578.533} C_VEL
LIN {X 0,Y 447.156,Z 281.74,A -85,B 0,C 180,E1 -8579.084,E2 -8579.084} C_VEL
LIN {X 0,Y 445.59,Z 275.379,A -85,B 0,C 180,E1 -8579.349,E2 -8579.349} C_VEL
LIN {X 0,Y 445.705,Z 270.868,A -85,B 0,C 180,E1 -8582.419,E2 -8582.419} C_VEL
LIN {X 0,Y 445.844,Z 266.178,A -85,B 0,C 180,E1 -8585.678,E2 -8585.678} C_VEL
LIN {X 0,Y 446.004,Z 261.433,A -85,B 0,C 180,E1 -8589.072,E2 -8589.072} C_VEL
LIN {X 0,Y 446.167,Z 256.592,A -85,B 0,C 180,E1 -8592.634,E2 -8592.634} C_VEL
LIN {X 0,Y 446.369,Z 253.303,A -85,B 0,C 180,E1 -8595.113,E2 -8595.113} C_VEL
LIN {X 0,Y 446.435,Z 249.948,A -85,B 0,C 180,E1 -8597.721,E2 -8597.721} C_VEL
LIN {X 0,Y 446.396,Z 248.25,A -85,B 0,C 180,E1 -8599.085,E2 -8599.085} C_VEL
LIN {X 0,Y 446.398,Z 247.887,A -85,B 0,C 180,E1 -8600.482,E2 -8600.482} C_VEL
LIN {X 0,Y 446.395,Z 247.881,A -85,B 0,C 180,E1 -8603.41,E2 -8603.41} C_VEL
LIN {X 0,Y 446.435,Z 247.878,A -85,B 0,C 180,E1 -8606.567,E2 -8606.567} C_VEL
LIN {X 0,Y 446.428,Z 247.878,A -85,B 0,C 180,E1 -8609.977,E2 -8609.977} C_VEL
LIN {X 0,Y 446.462,Z 247.872,A -85,B 0,C 180,E1 -8612.84,E2 -8612.84} C_VEL
LIN {X 0,Y 446.454,Z 247.873,A -85,B 0,C 180,E1 -8615.924,E2 -8615.924} C_VEL
LIN {X 0,Y 446.484,Z 247.869,A -85,B 0,C 180,E1 -8618.776,E2 -8618.776} C_VEL
LIN {X 0,Y 446.445,Z 247.873,A -85,B 0,C 180,E1 -8621.65,E2 -8621.65} C_VEL
LIN {X 0,Y 446.504,Z 247.866,A -85,B 0,C 180,E1 -8624.481,E2 -8624.481} C_VEL
LIN {X 0,Y 446.506,Z 247.868,A -85,B 0,C 180,E1 -8628.194,E2 -8628.194} C_VEL
LIN {X 0,Y 446.59,Z 247.856,A -85,B 0,C 180,E1 -8631.859,E2 -8631.859} C_VEL
LIN {X 0,Y 446.629,Z 247.853,A -85,B 0,C 180,E1 -8634.584,E2 -8634.584} C_VEL
LIN {X 0,Y 446.701,Z 247.844,A -85,B 0,C 180,E1 -8637.296,E2 -8637.296} C_VEL
LIN {X 0,Y 446.78,Z 247.831,A -85,B 0,C 180,E1 -8640.001,E2 -8640.001} C_VEL
LIN {X 0,Y 446.701,Z 247.842,A -85,B 0,C 180,E1 -8642.706,E2 -8642.706} C_VEL
LIN {X 0,Y 446.629,Z 247.852,A -85,B 0,C 180,E1 -8646.325,E2 -8646.325} C_VEL
LIN {X 0,Y 446.53,Z 247.864,A -85,B 0,C 180,E1 -8649.057,E2 -8649.057} C_VEL
LIN {X 0,Y 446.513,Z 247.868,A -85,B 0,C 180,E1 -8652.731,E2 -8652.731} C_VEL
LIN {X 0,Y 446.483,Z 247.87,A -85,B 0,C 180,E1 -8656.46,E2 -8656.46} C_VEL
LIN {X 0,Y 446.462,Z 247.873,A -85,B 0,C 180,E1 -8659.304,E2 -8659.304} C_VEL
LIN {X 0,Y 446.411,Z 247.881,A -85,B 0,C 180,E1 -8662.201,E2 -8662.201} C_VEL
LIN {X 0,Y 446.444,Z 247.877,A -85,B 0,C 180,E1 -8665.154,E2 -8665.154} C_VEL
LIN {X 0,Y 446.443,Z 247.877,A -85,B 0,C 180,E1 -8668.182,E2 -8668.182} C_VEL
LIN {X 0,Y 446.411,Z 247.88,A -85,B 0,C 180,E1 -8671.302,E2 -8671.302} C_VEL
LIN {X 0,Y 446.424,Z 247.877,A -85,B 0,C 180,E1 -8674.524,E2 -8674.524} C_VEL
LIN {X 0,Y 446.412,Z 247.88,A -85,B 0,C 180,E1 -8678.08,E2 -8678.08} C_VEL
LIN {X 0,Y 446.424,Z 247.875,A -85,B 0,C 180,E1 -8680.919,E2 -8680.919} C_VEL
LIN {X 0,Y 446.398,Z 247.881,A -85,B 0,C 180,E1 -8683.847,E2 -8683.847} C_VEL
LIN {X 0,Y 446.385,Z 247.885,A -85,B 0,C 180,E1 -8686.406,E2 -8686.406} C_VEL
LIN {X 0,Y 446.466,Z 248.081,A -85,B 0,C 180,E1 -8689.451,E2 -8689.451} C_VEL
LIN {X 0,Y 447.234,Z 252.676,A -85,B 0,C 180,E1 -8692.204,E2 -8692.204} C_VEL
LIN {X 0,Y 447.625,Z 257.236,A -85,B 0,C 180,E1 -8694.73,E2 -8694.73} C_VEL
LIN {X 0,Y 447.387,Z 261.971,A -85,B 0,C 180,E1 -8697.184,E2 -8697.184} C_VEL
LIN {X 0,Y 447.008,Z 268.327,A -85,B 0,C 180,E1 -8700.335,E2 -8700.335} C_VEL
LIN {X 0,Y 446.507,Z 275.721,A -85,B 0,C 180,E1 -8703.851,E2 -8703.851} C_VEL
LIN {X 0,Y 446.249,Z 282.139,A -85,B 0,C 180,E1 -8706.814,E2 -8706.814} C_VEL
LIN {X 0,Y 446.025,Z 288.622,A -85,B 0,C 180,E1 -8709.718,E2 -8709.718} C_VEL
LIN {X 0,Y 445.826,Z 296.19,A -85,B 0,C 180,E1 -8713.045,E2 -8713.045} C_VEL
LIN {X 0,Y 445.771,Z 297.811,A -85,B 0,C 180,E1 -8713.711,E2 -8713.711} C_VEL
LIN {X 0,Y 448.155,Z 310.811,A -85,B 0,C 180,E1 -8714.175,E2 -8714.175} C_VEL
LIN {X 0,Y 449.489,Z 322.028,A -85,B 0,C 180,E1 -8714.702,E2 -8714.702} C_VEL
LIN {X 0,Y 448.847,Z 334.202,A -85,B 0,C 180,E1 -8715.376,E2 -8715.376} C_VEL
LIN {X 0,Y 448.145,Z 346.624,A -85,B 0,C 180,E1 -8716.279,E2 -8716.279} C_VEL
LIN {X 0,Y 447.538,Z 357.53,A -85,B 0,C 180,E1 -8717.3,E2 -8717.3} C_VEL
LIN {X 0,Y 447.019,Z 367.318,A -85,B 0,C 180,E1 -8718.437,E2 -8718.437} C_VEL
LIN {X 0,Y 446.438,Z 375.356,A -85,B 0,C 180,E1 -8719.57,E2 -8719.57} C_VEL
LIN {X 0,Y 446.026,Z 383.265,A -85,B 0,C 180,E1 -8720.934,E2 -8720.934} C_VEL
LIN {X 0,Y 445.737,Z 389.593,A -85,B 0,C 180,E1 -8722.298,E2 -8722.298} C_VEL
LIN {X 0,Y 445.488,Z 395.508,A -85,B 0,C 180,E1 -8723.937,E2 -8723.937} C_VEL
LIN {X 0,Y 445.413,Z 399.624,A -85,B 0,C 180,E1 -8725.475,E2 -8725.475} C_VEL
LIN {X 0,Y 445.378,Z 401.446,A -85,B 0,C 180,E1 -8726.381,E2 -8726.381} C_VEL
LIN {X 0,Y 445.434,Z 402.818,A -85,B 0,C 180,E1 -8727.287,E2 -8727.287} C_VEL
LIN {X 0,Y 445.339,Z 404.385,A -85,B 0,C 180,E1 -8729.096,E2 -8729.096} C_VEL
LIN {X 0,Y 445.343,Z 404.569,A -85,B 0,C 180,E1 -8730,E2 -8730} C_VEL
LIN {X 0,Y 445.357,Z 403.702,A -85,B 0,C 180,E1 -8731.809,E2 -8731.809} C_VEL
LIN {X 0,Y 445.434,Z 402.689,A -85,B 0,C 180,E1 -8732.713,E2 -8732.713} C_VEL
LIN {X 0,Y 445.38,Z 401.252,A -85,B 0,C 180,E1 -8733.619,E2 -8733.619} C_VEL
LIN {X 0,Y 445.475,Z 398.275,A -85,B 0,C 180,E1 -8734.978,E2 -8734.978} C_VEL
LIN {X 0,Y 445.559,Z 392.784,A -85,B 0,C 180,E1 -8736.748,E2 -8736.748} C_VEL
LIN {X 0,Y 445.794,Z 387.014,A -85,B 0,C 180,E1 -8738.157,E2 -8738.157} C_VEL
LIN {X 0,Y 446.148,Z 380.005,A -85,B 0,C 180,E1 -8739.52,E2 -8739.52} C_VEL
LIN {X 0,Y 446.565,Z 371.211,A -85,B 0,C 180,E1 -8740.886,E2 -8740.886} C_VEL
LIN {X 0,Y 447.182,Z 361.225,A -85,B 0,C 180,E1 -8742.134,E2 -8742.134} C_VEL
LIN {X 0,Y 447.683,Z 350.807,A -85,B 0,C 180,E1 -8743.179,E2 -8743.179} C_VEL
LIN {X 0,Y 448.241,Z 339.742,A -85,B 0,C 180,E1 -8744.065,E2 -8744.065} C_VEL
LIN {X 0,Y 448.879,Z 328.034,A -85,B 0,C 180,E1 -8744.797,E2 -8744.797} C_VEL
LIN {X 0,Y 449.02,Z 319.997,A -85,B 0,C 180,E1 -8745.198,E2 -8745.198} C_VEL
LIN {X 0,Y 447.111,Z 306.732,A -85,B 0,C 180,E1 -8745.758,E2 -8745.758} C_VEL
LIN {X 0,Y 445.706,Z 297.833,A -85,B 0,C 180,E1 -8746.05,E2 -8746.05} C_VEL
LIN {X 0,Y 445.906,Z 290.18,A -85,B 0,C 180,E1 -8749.328,E2 -8749.328} C_VEL
LIN {X 0,Y 446.157,Z 283.54,A -85,B 0,C 180,E1 -8752.213,E2 -8752.213} C_VEL
LIN {X 0,Y 446.425,Z 275.77,A -85,B 0,C 180,E1 -8755.653,E2 -8755.653} C_VEL
LIN {X 0,Y 446.738,Z 267.985,A -85,B 0,C 180,E1 -8759.188,E2 -8759.188} C_VEL
LIN {X 0,Y 447.117,Z 261.331,A -85,B 0,C 180,E1 -8762.304,E2 -8762.304} C_VEL
LIN {X 0,Y 447.372,Z 255.287,A -85,B 0,C 180,E1 -8765.224,E2 -8765.224} C_VEL
LIN {X 0,Y 447.009,Z 251.319,A -85,B 0,C 180,E1 -8767.249,E2 -8767.249} C_VEL
LIN {X 0,Y 446.468,Z 247.875,A -85,B 0,C 180,E1 -8769.148,E2 -8769.148} C_VEL
LIN {X 0,Y 446.37,Z 247.886,A -85,B 0,C 180,E1 -8772.61,E2 -8772.61} C_VEL
LIN {X 0,Y 446.41,Z 247.879,A -85,B 0,C 180,E1 -8775.108,E2 -8775.108} C_VEL
LIN {X 0,Y 446.396,Z 247.882,A -85,B 0,C 180,E1 -8778.604,E2 -8778.604} C_VEL
LIN {X 0,Y 446.392,Z 247.879,A -85,B 0,C 180,E1 -8781.923,E2 -8781.923} C_VEL
LIN {X 0,Y 446.416,Z 247.876,A -85,B 0,C 180,E1 -8785.475,E2 -8785.475} C_VEL
LIN {X 0,Y 446.41,Z 247.878,A -85,B 0,C 180,E1 -8788.698,E2 -8788.698} C_VEL
LIN {X 0,Y 446.442,Z 247.874,A -85,B 0,C 180,E1 -8791.829,E2 -8791.829} C_VEL
LIN {X 0,Y 446.432,Z 247.874,A -85,B 0,C 180,E1 -8794.845,E2 -8794.845} C_VEL
LIN {X 0,Y 446.442,Z 247.875,A -85,B 0,C 180,E1 -8798.244,E2 -8798.244} C_VEL
LIN {X 0,Y 446.445,Z 247.874,A -85,B 0,C 180,E1 -8801.648,E2 -8801.648} C_VEL
LIN {X 0,Y 446.5,Z 247.866,A -85,B 0,C 180,E1 -8804.479,E2 -8804.479} C_VEL
LIN {X 0,Y 446.51,Z 247.865,A -85,B 0,C 180,E1 -8808.192,E2 -8808.192} C_VEL
LIN {X 0,Y 446.592,Z 247.856,A -85,B 0,C 180,E1 -8811.857,E2 -8811.857} C_VEL
LIN {X 0,Y 446.636,Z 247.852,A -85,B 0,C 180,E1 -8814.581,E2 -8814.581} C_VEL
LIN {X 0,Y 446.699,Z 247.843,A -85,B 0,C 180,E1 -8817.294,E2 -8817.294} C_VEL
LIN {X 0,Y 446.785,Z 247.831,A -85,B 0,C 180,E1 -8819.999,E2 -8819.999} C_VEL
LIN {X 0,Y 446.7,Z 247.842,A -85,B 0,C 180,E1 -8822.704,E2 -8822.704} C_VEL
LIN {X 0,Y 446.639,Z 247.851,A -85,B 0,C 180,E1 -8826.323,E2 -8826.323} C_VEL
LIN {X 0,Y 446.529,Z 247.864,A -85,B 0,C 180,E1 -8829.054,E2 -8829.054} C_VEL
LIN {X 0,Y 446.511,Z 247.865,A -85,B 0,C 180,E1 -8832.729,E2 -8832.729} C_VEL
LIN {X 0,Y 446.485,Z 247.869,A -85,B 0,C 180,E1 -8836.227,E2 -8836.227} C_VEL
LIN {X 0,Y 446.458,Z 247.872,A -85,B 0,C 180,E1 -8839.302,E2 -8839.302} C_VEL
LIN {X 0,Y 446.407,Z 247.878,A -85,B 0,C 180,E1 -8842.199,E2 -8842.199} C_VEL
LIN {X 0,Y 446.446,Z 247.873,A -85,B 0,C 180,E1 -8845.152,E2 -8845.152} C_VEL
LIN {X 0,Y 446.472,Z 247.869,A -85,B 0,C 180,E1 -8848.178,E2 -8848.178} C_VEL
LIN {X 0,Y 446.408,Z 247.882,A -85,B 0,C 180,E1 -8851.299,E2 -8851.299} C_VEL
LIN {X 0,Y 446.418,Z 247.875,A -85,B 0,C 180,E1 -8854.522,E2 -8854.522} C_VEL
LIN {X 0,Y 446.426,Z 247.873,A -85,B 0,C 180,E1 -8858.083,E2 -8858.083} C_VEL
LIN {X 0,Y 446.436,Z 247.878,A -85,B 0,C 180,E1 -8860.92,E2 -8860.92} C_VEL
LIN {X 0,Y 446.433,Z 247.872,A -85,B 0,C 180,E1 -8863.84,E2 -8863.84} C_VEL
LIN {X 0,Y 446.408,Z 247.877,A -85,B 0,C 180,E1 -8866.4,E2 -8866.4} C_VEL
LIN {X 0,Y 446.435,Z 247.872,A -85,B 0,C 180,E1 -8869.802,E2 -8869.802} C_VEL
LIN {X 0,Y 446.415,Z 247.876,A -85,B 0,C 180,E1 -8872.123,E2 -8872.123} C_VEL
LIN {X 0,Y 446.417,Z 247.874,A -85,B 0,C 180,E1 -8875.477,E2 -8875.477} C_VEL
LIN {X 0,Y 446.403,Z 247.879,A -85,B 0,C 180,E1 -8878.699,E2 -8878.699} C_VEL
LIN {X 0,Y 446.472,Z 247.87,A -85,B 0,C 180,E1 -8881.821,E2 -8881.821} C_VEL
LIN {X 0,Y 446.426,Z 247.874,A -85,B 0,C 180,E1 -8884.846,E2 -8884.846} C_VEL
LIN {X 0,Y 446.287,Z 247.894,A -85,B 0,C 180,E1 -8887.794,E2 -8887.794} C_VEL
LIN {X 0,Y 446.237,Z 248.028,A -85,B 0,C 180,E1 -8888.309,E2 -8888.309} C_VEL
LIN {X 0,Y 446.201,Z 252.633,A -85,B 0,C 180,E1 -8891.639,E2 -8891.639} C_VEL
LIN {X 0,Y 446.089,Z 256.637,A -85,B 0,C 180,E1 -8894.465,E2 -8894.465} C_VEL
LIN {X 0,Y 446.002,Z 261.992,A -85,B 0,C 180,E1 -8898.179,E2 -8898.179} C_VEL
LIN {X 0,Y 445.877,Z 267.386,A -85,B 0,C 180,E1 -8901.845,E2 -8901.845} C_VEL
LIN {X 0,Y 445.879,Z 270.103,A -85,B 0,C 180,E1 -8903.665,E2 -8903.665} C_VEL
LIN {X 0,Y 445.76,Z 274.598,A -85,B 0,C 180,E1 -8906.631,E2 -8906.631} C_VEL
LIN {X 0,Y 445.74,Z 275.838,A -85,B 0,C 180,E1 -8906.891,E2 -8906.891} C_VEL
LIN {X 0,Y 445.695,Z 278.928,A -85,B 0,C 180,E1 -8907.116,E2 -8907.116} C_VEL
LIN {X 0,Y 445.099,Z 289.549,A -85,B 0,C 180,E1 -8907.474,E2 -8907.474} C_VEL
LIN {X 0,Y 442.667,Z 300.575,A -85,B 0,C 180,E1 -8907.885,E2 -8907.885} C_VEL
LIN {X 0,Y 442.121,Z 304.166,A -85,B 0,C 180,E1 -8908.085,E2 -8908.085} C_VEL
LIN {X 0,Y 441.6,Z 316.115,A -85,B 0,C 180,E1 -8908.86,E2 -8908.86} C_VEL
LIN {X 0,Y 441.013,Z 327.125,A -85,B 0,C 180,E1 -8909.772,E2 -8909.772} C_VEL
LIN {X 0,Y 440.458,Z 336.065,A -85,B 0,C 180,E1 -8910.686,E2 -8910.686} C_VEL
LIN {X 0,Y 439.928,Z 345.238,A -85,B 0,C 180,E1 -8911.831,E2 -8911.831} C_VEL
LIN {X 0,Y 439.351,Z 354.175,A -85,B 0,C 180,E1 -8913.209,E2 -8913.209} C_VEL
LIN {X 0,Y 439.003,Z 361.372,A -85,B 0,C 180,E1 -8914.591,E2 -8914.591} C_VEL
LIN {X 0,Y 438.735,Z 367.138,A -85,B 0,C 180,E1 -8915.976,E2 -8915.976} C_VEL
LIN {X 0,Y 438.561,Z 371.683,A -85,B 0,C 180,E1 -8917.365,E2 -8917.365} C_VEL
LIN {X 0,Y 438.418,Z 374.088,A -85,B 0,C 180,E1 -8918.295,E2 -8918.295} C_VEL
LIN {X 0,Y 438.316,Z 376.06,A -85,B 0,C 180,E1 -8919.226,E2 -8919.226} C_VEL
LIN {X 0,Y 438.26,Z 377.613,A -85,B 0,C 180,E1 -8920.16,E2 -8920.16} C_VEL
LIN {X 0,Y 438.257,Z 379.368,A -85,B 0,C 180,E1 -8921.991,E2 -8921.991} C_VEL
LIN {X 0,Y 438.187,Z 379.687,A -85,B 0,C 180,E1 -8922.976,E2 -8922.976} C_VEL
LIN {X 0,Y 438.158,Z 379.573,A -85,B 0,C 180,E1 -8923.921,E2 -8923.921} C_VEL
LIN {X 0,Y 438.199,Z 379.003,A -85,B 0,C 180,E1 -8924.869,E2 -8924.869} C_VEL
LIN {X 0,Y 438.266,Z 378.027,A -85,B 0,C 180,E1 -8925.819,E2 -8925.819} C_VEL
LIN {X 0,Y 438.266,Z 376.635,A -85,B 0,C 180,E1 -8926.776,E2 -8926.776} C_VEL
LIN {X 0,Y 438.487,Z 373.651,A -85,B 0,C 180,E1 -8928.212,E2 -8928.212} C_VEL
LIN {X 0,Y 438.681,Z 369.536,A -85,B 0,C 180,E1 -8929.659,E2 -8929.659} C_VEL
LIN {X 0,Y 439.045,Z 363.083,A -85,B 0,C 180,E1 -8931.356,E2 -8931.356} C_VEL
LIN {X 0,Y 439.513,Z 355.967,A -85,B 0,C 180,E1 -8932.815,E2 -8932.815} C_VEL
LIN {X 0,Y 440.109,Z 347.419,A -85,B 0,C 180,E1 -8934.207,E2 -8934.207} C_VEL
LIN {X 0,Y 440.75,Z 337.52,A -85,B 0,C 180,E1 -8935.501,E2 -8935.501} C_VEL
LIN {X 0,Y 441.333,Z 328.295,A -85,B 0,C 180,E1 -8936.479,E2 -8936.479} C_VEL
LIN {X 0,Y 441.914,Z 318.737,A -85,B 0,C 180,E1 -8937.31,E2 -8937.31} C_VEL
LIN {X 0,Y 442.548,Z 306.906,A -85,B 0,C 180,E1 -8938.128,E2 -8938.128} C_VEL
LIN {X 0,Y 443.013,Z 296.621,A -85,B 0,C 180,E1 -8938.678,E2 -8938.678} C_VEL
LIN {X 0,Y 440.939,Z 285.398,A -85,B 0,C 180,E1 -8939.234,E2 -8939.234} C_VEL
LIN {X 0,Y 438.539,Z 275.6,A -85,B 0,C 180,E1 -8939.644,E2 -8939.644} C_VEL
LIN {X 0,Y 438.659,Z 270.735,A -85,B 0,C 180,E1 -8943.005,E2 -8943.005} C_VEL
LIN {X 0,Y 438.767,Z 267.599,A -85,B 0,C 180,E1 -8945.227,E2 -8945.227} C_VEL
LIN {X 0,Y 438.929,Z 262.852,A -85,B 0,C 180,E1 -8948.641,E2 -8948.641} C_VEL
LIN {X 0,Y 439.093,Z 258.021,A -85,B 0,C 180,E1 -8952.239,E2 -8952.239} C_VEL
LIN {X 0,Y 439.357,Z 254.073,A -85,B 0,C 180,E1 -8955.267,E2 -8955.267} C_VEL
LIN {X 0,Y 439.419,Z 250.861,A -85,B 0,C 180,E1 -8957.8,E2 -8957.8} C_VEL
LIN {X 0,Y 439.372,Z 249.373,A -85,B 0,C 180,E1 -8959.02,E2 -8959.02} C_VEL
LIN {X 0,Y 439.344,Z 248.766,A -85,B 0,C 180,E1 -8960.22,E2 -8960.22} C_VEL
LIN {X 0,Y 439.344,Z 248.761,A -85,B 0,C 180,E1 -8963.112,E2 -8963.112} C_VEL
LIN {X 0,Y 439.384,Z 248.757,A -85,B 0,C 180,E1 -8966.276,E2 -8966.276} C_VEL
LIN {X 0,Y 439.401,Z 248.752,A -85,B 0,C 180,E1 -8969.733,E2 -8969.733} C_VEL
LIN {X 0,Y 439.428,Z 248.748,A -85,B 0,C 180,E1 -8972.368,E2 -8972.368} C_VEL
LIN {X 0,Y 439.404,Z 248.751,A -85,B 0,C 180,E1 -8975.735,E2 -8975.735} C_VEL
LIN {X 0,Y 439.439,Z 248.747,A -85,B 0,C 180,E1 -8978.419,E2 -8978.419} C_VEL
LIN {X 0,Y 439.416,Z 248.749,A -85,B 0,C 180,E1 -8981.346,E2 -8981.346} C_VEL
LIN {X 0,Y 439.463,Z 248.744,A -85,B 0,C 180,E1 -8984.226,E2 -8984.226} C_VEL
LIN {X 0,Y 439.472,Z 248.743,A -85,B 0,C 180,E1 -8988.002,E2 -8988.002} C_VEL
LIN {X 0,Y 439.537,Z 248.735,A -85,B 0,C 180,E1 -8991.727,E2 -8991.727} C_VEL
LIN {X 0,Y 439.604,Z 248.729,A -85,B 0,C 180,E1 -8994.497,E2 -8994.497} C_VEL
LIN {X 0,Y 439.627,Z 248.723,A -85,B 0,C 180,E1 -8998.169,E2 -8998.169} C_VEL
LIN {X 0,Y 439.75,Z 248.707,A -85,B 0,C 180,E1 -9000.001,E2 -9000.001} C_VEL
LIN {X 0,Y 439.648,Z 248.72,A -85,B 0,C 180,E1 -9002.75,E2 -9002.75} C_VEL
LIN {X 0,Y 439.604,Z 248.728,A -85,B 0,C 180,E1 -9006.426,E2 -9006.426} C_VEL
LIN {X 0,Y 439.492,Z 248.741,A -85,B 0,C 180,E1 -9009.203,E2 -9009.203} C_VEL
LIN {X 0,Y 439.458,Z 248.745,A -85,B 0,C 180,E1 -9012.939,E2 -9012.939} C_VEL
LIN {X 0,Y 439.44,Z 248.748,A -85,B 0,C 180,E1 -9016.35,E2 -9016.35} C_VEL
LIN {X 0,Y 439.396,Z 248.754,A -85,B 0,C 180,E1 -9019.628,E2 -9019.628} C_VEL
LIN {X 0,Y 439.359,Z 248.759,A -85,B 0,C 180,E1 -9022.577,E2 -9022.577} C_VEL
LIN {X 0,Y 439.387,Z 248.756,A -85,B 0,C 180,E1 -9025.587,E2 -9025.587} C_VEL
LIN {X 0,Y 439.394,Z 248.755,A -85,B 0,C 180,E1 -9028.676,E2 -9028.676} C_VEL
LIN {X 0,Y 439.366,Z 248.76,A -85,B 0,C 180,E1 -9032.032,E2 -9032.032} C_VEL
LIN {X 0,Y 439.39,Z 248.756,A -85,B 0,C 180,E1 -9035.341,E2 -9035.341} C_VEL
LIN {X 0,Y 439.375,Z 248.755,A -85,B 0,C 180,E1 -9038.597,E2 -9038.597} C_VEL
LIN {X 0,Y 439.386,Z 248.755,A -85,B 0,C 180,E1 -9041.258,E2 -9041.258} C_VEL
LIN {X 0,Y 439.397,Z 248.746,A -85,B 0,C 180,E1 -9044.731,E2 -9044.731} C_VEL
LIN {X 0,Y 439.349,Z 248.763,A -85,B 0,C 180,E1 -9047.791,E2 -9047.791} C_VEL
LIN {X 0,Y 439.356,Z 248.775,A -85,B 0,C 180,E1 -9049.018,E2 -9049.018} C_VEL
LIN {X 0,Y 440.078,Z 252.799,A -85,B 0,C 180,E1 -9051.493,E2 -9051.493} C_VEL
LIN {X 0,Y 440.595,Z 256.832,A -85,B 0,C 180,E1 -9053.83,E2 -9053.83} C_VEL
LIN {X 0,Y 440.561,Z 260.96,A -85,B 0,C 180,E1 -9056.06,E2 -9056.06} C_VEL
LIN {X 0,Y 440.061,Z 267.856,A -85,B 0,C 180,E1 -9059.589,E2 -9059.589} C_VEL
LIN {X 0,Y 439.654,Z 273.549,A -85,B 0,C 180,E1 -9062.383,E2 -9062.383} C_VEL
LIN {X 0,Y 439.31,Z 280.674,A -85,B 0,C 180,E1 -9065.767,E2 -9065.767} C_VEL
LIN {X 0,Y 439.046,Z 287.445,A -85,B 0,C 180,E1 -9068.89,E2 -9068.89} C_VEL
LIN {X 0,Y 438.753,Z 294.993,A -85,B 0,C 180,E1 -9072.282,E2 -9072.282} C_VEL
LIN {X 0,Y 438.728,Z 297.491,A -85,B 0,C 180,E1 -9073.393,E2 -9073.393} C_VEL
LIN {X 0,Y 441.305,Z 311.642,A -85,B 0,C 180,E1 -9073.93,E2 -9073.93} C_VEL
LIN {X 0,Y 442.636,Z 322.432,A -85,B 0,C 180,E1 -9074.459,E2 -9074.459} C_VEL
LIN {X 0,Y 441.995,Z 334.465,A -85,B 0,C 180,E1 -9075.144,E2 -9075.144} C_VEL
LIN {X 0,Y 441.257,Z 346.777,A -85,B 0,C 180,E1 -9076.061,E2 -9076.061} C_VEL
LIN {X 0,Y 440.603,Z 357.597,A -85,B 0,C 180,E1 -9077.097,E2 -9077.097} C_VEL
LIN {X 0,Y 440.056,Z 367.333,A -85,B 0,C 180,E1 -9078.251,E2 -9078.251} C_VEL
LIN {X 0,Y 439.432,Z 375.334,A -85,B 0,C 180,E1 -9079.402,E2 -9079.402} C_VEL
LIN {X 0,Y 438.993,Z 383.199,A -85,B 0,C 180,E1 -9080.788,E2 -9080.788} C_VEL
LIN {X 0,Y 438.691,Z 389.494,A -85,B 0,C 180,E1 -9082.174,E2 -9082.174} C_VEL
LIN {X 0,Y 438.464,Z 394.675,A -85,B 0,C 180,E1 -9083.61,E2 -9083.61} C_VEL
LIN {X 0,Y 438.385,Z 398.41,A -85,B 0,C 180,E1 -9084.942,E2 -9084.942} C_VEL
LIN {X 0,Y 438.28,Z 401.283,A -85,B 0,C 180,E1 -9086.323,E2 -9086.323} C_VEL
LIN {X 0,Y 438.342,Z 402.647,A -85,B 0,C 180,E1 -9087.243,E2 -9087.243} C_VEL
LIN {X 0,Y 438.253,Z 404.198,A -85,B 0,C 180,E1 -9089.081,E2 -9089.081} C_VEL
LIN {X 0,Y 438.254,Z 404.364,A -85,B 0,C 180,E1 -9090,E2 -9090} C_VEL
LIN {X 0,Y 438.279,Z 403.482,A -85,B 0,C 180,E1 -9091.838,E2 -9091.838} C_VEL
LIN {X 0,Y 438.342,Z 402.459,A -85,B 0,C 180,E1 -9092.757,E2 -9092.757} C_VEL
LIN {X 0,Y 438.282,Z 401.004,A -85,B 0,C 180,E1 -9093.678,E2 -9093.678} C_VEL
LIN {X 0,Y 438.385,Z 398.011,A -85,B 0,C 180,E1 -9095.058,E2 -9095.058} C_VEL
LIN {X 0,Y 438.451,Z 393.957,A -85,B 0,C 180,E1 -9096.442,E2 -9096.442} C_VEL
LIN {X 0,Y 438.69,Z 387.717,A -85,B 0,C 180,E1 -9098.058,E2 -9098.058} C_VEL
LIN {X 0,Y 439.033,Z 380.917,A -85,B 0,C 180,E1 -9099.444,E2 -9099.444} C_VEL
LIN {X 0,Y 439.448,Z 372.457,A -85,B 0,C 180,E1 -9100.831,E2 -9100.831} C_VEL
LIN {X 0,Y 440.02,Z 363.737,A -85,B 0,C 180,E1 -9101.984,E2 -9101.984} C_VEL
LIN {X 0,Y 440.544,Z 353.856,A -85,B 0,C 180,E1 -9103.054,E2 -9103.054} C_VEL
LIN {X 0,Y 441.173,Z 342.3,A -85,B 0,C 180,E1 -9104.06,E2 -9104.06} C_VEL
LIN {X 0,Y 441.809,Z 330.331,A -85,B 0,C 180,E1 -9104.862,E2 -9104.862} C_VEL
LIN {X 0,Y 442.023,Z 320.442,A -85,B 0,C 180,E1 -9105.386,E2 -9105.386} C_VEL
LIN {X 0,Y 440.106,Z 306.848,A -85,B 0,C 180,E1 -9105.974,E2 -9105.974} C_VEL
LIN {X 0,Y 438.614,Z 297.678,A -85,B 0,C 180,E1 -9106.272,E2 -9106.272} C_VEL
LIN {X 0,Y 438.847,Z 289.928,A -85,B 0,C 180,E1 -9109.652,E2 -9109.652} C_VEL
LIN {X 0,Y 439.069,Z 283.293,A -85,B 0,C 180,E1 -9112.591,E2 -9112.591} C_VEL
LIN {X 0,Y 439.345,Z 276.642,A -85,B 0,C 180,E1 -9115.588,E2 -9115.588} C_VEL
LIN {X 0,Y 439.698,Z 268.866,A -85,B 0,C 180,E1 -9119.176,E2 -9119.176} C_VEL
LIN {X 0,Y 440.068,Z 262.555,A -85,B 0,C 180,E1 -9122.174,E2 -9122.174} C_VEL
LIN {X 0,Y 440.328,Z 256.661,A -85,B 0,C 180,E1 -9125.07,E2 -9125.07} C_VEL
LIN {X 0,Y 440.07,Z 252.878,A -85,B 0,C 180,E1 -9127.011,E2 -9127.011} C_VEL
LIN {X 0,Y 439.419,Z 248.752,A -85,B 0,C 180,E1 -9129.327,E2 -9129.327} C_VEL
LIN {X 0,Y 439.327,Z 248.763,A -85,B 0,C 180,E1 -9132.618,E2 -9132.618} C_VEL
LIN {X 0,Y 439.364,Z 248.755,A -85,B 0,C 180,E1 -9135.265,E2 -9135.265} C_VEL
LIN {X 0,Y 439.359,Z 248.76,A -85,B 0,C 180,E1 -9138.746,E2 -9138.746} C_VEL
LIN {X 0,Y 439.351,Z 248.756,A -85,B 0,C 180,E1 -9141.61,E2 -9141.61} C_VEL
LIN {X 0,Y 439.387,Z 248.753,A -85,B 0,C 180,E1 -9144.842,E2 -9144.842} C_VEL
LIN {X 0,Y 439.367,Z 248.756,A -85,B 0,C 180,E1 -9148.138,E2 -9148.138} C_VEL
LIN {X 0,Y 439.396,Z 248.751,A -85,B 0,C 180,E1 -9151.605,E2 -9151.605} C_VEL
LIN {X 0,Y 439.37,Z 248.756,A -85,B 0,C 180,E1 -9154.412,E2 -9154.412} C_VEL
LIN {X 0,Y 439.357,Z 248.756,A -85,B 0,C 180,E1 -9157.423,E2 -9157.423} C_VEL
LIN {X 0,Y 439.434,Z 248.747,A -85,B 0,C 180,E1 -9160.662,E2 -9160.662} C_VEL
LIN {X 0,Y 439.455,Z 248.745,A -85,B 0,C 180,E1 -9164.223,E2 -9164.223} C_VEL
LIN {X 0,Y 439.476,Z 248.742,A -85,B 0,C 180,E1 -9168,E2 -9168} C_VEL
LIN {X 0,Y 439.54,Z 248.735,A -85,B 0,C 180,E1 -9171.725,E2 -9171.725} C_VEL
LIN {X 0,Y 439.611,Z 248.726,A -85,B 0,C 180,E1 -9174.495,E2 -9174.495} C_VEL
LIN {X 0,Y 439.626,Z 248.724,A -85,B 0,C 180,E1 -9178.167,E2 -9178.167} C_VEL
LIN {X 0,Y 439.755,Z 248.707,A -85,B 0,C 180,E1 -9179.999,E2 -9179.999} C_VEL
LIN {X 0,Y 439.647,Z 248.72,A -85,B 0,C 180,E1 -9182.748,E2 -9182.748} C_VEL
LIN {X 0,Y 439.61,Z 248.726,A -85,B 0,C 180,E1 -9186.424,E2 -9186.424} C_VEL
LIN {X 0,Y 439.491,Z 248.74,A -85,B 0,C 180,E1 -9189.201,E2 -9189.201} C_VEL
LIN {X 0,Y 439.455,Z 248.745,A -85,B 0,C 180,E1 -9192.937,E2 -9192.937} C_VEL
LIN {X 0,Y 439.436,Z 248.746,A -85,B 0,C 180,E1 -9196.348,E2 -9196.348} C_VEL
LIN {X 0,Y 439.391,Z 248.755,A -85,B 0,C 180,E1 -9199.625,E2 -9199.625} C_VEL
LIN {X 0,Y 439.354,Z 248.756,A -85,B 0,C 180,E1 -9202.575,E2 -9202.575} C_VEL
LIN {X 0,Y 439.394,Z 248.754,A -85,B 0,C 180,E1 -9205.584,E2 -9205.584} C_VEL
LIN {X 0,Y 439.413,Z 248.748,A -85,B 0,C 180,E1 -9208.672,E2 -9208.672} C_VEL
LIN {X 0,Y 439.362,Z 248.754,A -85,B 0,C 180,E1 -9211.86,E2 -9211.86} C_VEL
LIN {X 0,Y 439.389,Z 248.756,A -85,B 0,C 180,E1 -9215.155,E2 -9215.155} C_VEL
LIN {X 0,Y 439.387,Z 248.752,A -85,B 0,C 180,E1 -9218.593,E2 -9218.593} C_VEL
LIN {X 0,Y 439.393,Z 248.752,A -85,B 0,C 180,E1 -9221.259,E2 -9221.259} C_VEL
LIN {X 0,Y 439.397,Z 248.754,A -85,B 0,C 180,E1 -9224.728,E2 -9224.728} C_VEL
LIN {X 0,Y 439.385,Z 248.749,A -85,B 0,C 180,E1 -9227.796,E2 -9227.796} C_VEL
LIN {X 0,Y 439.417,Z 248.748,A -85,B 0,C 180,E1 -9230.227,E2 -9230.227} C_VEL
LIN {X 0,Y 439.364,Z 248.753,A -85,B 0,C 180,E1 -9233.713,E2 -9233.713} C_VEL
LIN {X 0,Y 439.36,Z 248.754,A -85,B 0,C 180,E1 -9237.054,E2 -9237.054} C_VEL
LIN {X 0,Y 439.37,Z 248.758,A -85,B 0,C 180,E1 -9240.274,E2 -9240.274} C_VEL
LIN {X 0,Y 439.406,Z 248.749,A -85,B 0,C 180,E1 -9243.395,E2 -9243.395} C_VEL
LIN {X 0,Y 439.326,Z 248.761,A -85,B 0,C 180,E1 -9246.427,E2 -9246.427} C_VEL
LIN {X 0,Y 439.194,Z 248.781,A -85,B 0,C 180,E1 -9248.139,E2 -9248.139} C_VEL
LIN {X 0,Y 439.164,Z 253.013,A -85,B 0,C 180,E1 -9251.334,E2 -9251.334} C_VEL
LIN {X 0,Y 439.022,Z 257.017,A -85,B 0,C 180,E1 -9254.209,E2 -9254.209} C_VEL
LIN {X 0,Y 438.955,Z 262.395,A -85,B 0,C 180,E1 -9257.987,E2 -9257.987} C_VEL
LIN {X 0,Y 438.812,Z 267.818,A -85,B 0,C 180,E1 -9261.712,E2 -9261.712} C_VEL
LIN {X 0,Y 438.815,Z 270.555,A -85,B 0,C 180,E1 -9263.563,E2 -9263.563} C_VEL
LIN {X 0,Y 438.693,Z 275.407,A -85,B 0,C 180,E1 -9266.814,E2 -9266.814} C_VEL
LIN {X 0,Y 441.295,Z 289.347,A -85,B 0,C 180,E1 -9267.347,E2 -9267.347} C_VEL
LIN {X 0,Y 442.484,Z 295.949,A -85,B 0,C 180,E1 -9267.667,E2 -9267.667} C_VEL
LIN {X 0,Y 442.121,Z 304.166,A -85,B 0,C 180,E1 -9268.085,E2 -9268.085} C_VEL
LIN {X 0,Y 441.236,Z 309.636,A -85,B 0,C 180,E1 -9268.392,E2 -9268.392} C_VEL
LIN {X 0,Y 437.939,Z 318.188,A -85,B 0,C 180,E1 -9268.906,E2 -9268.906} C_VEL
LIN {X 0,Y 434.676,Z 326.266,A -85,B 0,C 180,E1 -9269.508,E2 -9269.508} C_VEL
LIN {X 0,Y 433.828,Z 330.952,A -85,B 0,C 180,E1 -9269.947,E2 -9269.947} C_VEL
LIN {X 0,Y 433.245,Z 339.729,A -85,B 0,C 180,E1 -9270.929,E2 -9270.929} C_VEL
LIN {X 0,Y 432.733,Z 348.316,A -85,B 0,C 180,E1 -9272.094,E2 -9272.094} C_VEL
LIN {X 0,Y 432.165,Z 356.676,A -85,B 0,C 180,E1 -9273.496,E2 -9273.496} C_VEL
LIN {X 0,Y 431.758,Z 363.411,A -85,B 0,C 180,E1 -9274.902,E2 -9274.902} C_VEL
LIN {X 0,Y 431.568,Z 369.809,A -85,B 0,C 180,E1 -9276.614,E2 -9276.614} C_VEL
LIN {X 0,Y 431.397,Z 373.622,A -85,B 0,C 180,E1 -9277.959,E2 -9277.959} C_VEL
LIN {X 0,Y 431.204,Z 376.615,A -85,B 0,C 180,E1 -9279.38,E2 -9279.38} C_VEL
LIN {X 0,Y 431.156,Z 378.05,A -85,B 0,C 180,E1 -9280.329,E2 -9280.329} C_VEL
LIN {X 0,Y 431.164,Z 379.592,A -85,B 0,C 180,E1 -9282.048,E2 -9282.048} C_VEL
LIN {X 0,Y 431.079,Z 379.911,A -85,B 0,C 180,E1 -9283.193,E2 -9283.193} C_VEL
LIN {X 0,Y 431.062,Z 379.679,A -85,B 0,C 180,E1 -9284.155,E2 -9284.155} C_VEL
LIN {X 0,Y 431.194,Z 378.188,A -85,B 0,C 180,E1 -9285.928,E2 -9285.928} C_VEL
LIN {X 0,Y 431.217,Z 376.494,A -85,B 0,C 180,E1 -9287.059,E2 -9287.059} C_VEL
LIN {X 0,Y 431.462,Z 373.369,A -85,B 0,C 180,E1 -9288.519,E2 -9288.519} C_VEL
LIN {X 0,Y 431.672,Z 369.088,A -85,B 0,C 180,E1 -9289.992,E2 -9289.992} C_VEL
LIN {X 0,Y 432.007,Z 363.514,A -85,B 0,C 180,E1 -9291.471,E2 -9291.471} C_VEL
LIN {X 0,Y 432.501,Z 356.451,A -85,B 0,C 180,E1 -9292.953,E2 -9292.953} C_VEL
LIN {X 0,Y 433.159,Z 348.007,A -85,B 0,C 180,E1 -9294.365,E2 -9294.365} C_VEL
LIN {X 0,Y 433.832,Z 338.194,A -85,B 0,C 180,E1 -9295.679,E2 -9295.679} C_VEL
LIN {X 0,Y 434.531,Z 327.837,A -85,B 0,C 180,E1 -9296.797,E2 -9296.797} C_VEL
LIN {X 0,Y 435.211,Z 317.322,A -85,B 0,C 180,E1 -9297.702,E2 -9297.702} C_VEL
LIN {X 0,Y 435.864,Z 306.043,A -85,B 0,C 180,E1 -9298.468,E2 -9298.468} C_VEL
LIN {X 0,Y 436.215,Z 297.415,A -85,B 0,C 180,E1 -9298.939,E2 -9298.939} C_VEL
LIN {X 0,Y 433.987,Z 285.693,A -85,B 0,C 180,E1 -9299.538,E2 -9299.538} C_VEL
LIN {X 0,Y 431.523,Z 275.791,A -85,B 0,C 180,E1 -9299.966,E2 -9299.966} C_VEL
LIN {X 0,Y 431.648,Z 270.618,A -85,B 0,C 180,E1 -9303.612,E2 -9303.612} C_VEL
LIN {X 0,Y 431.77,Z 265.783,A -85,B 0,C 180,E1 -9307.103,E2 -9307.103} C_VEL
LIN {X 0,Y 431.926,Z 261.734,A -85,B 0,C 180,E1 -9310.118,E2 -9310.118} C_VEL
LIN {X 0,Y 432.12,Z 257.832,A -85,B 0,C 180,E1 -9313.084,E2 -9313.084} C_VEL
LIN {X 0,Y 432.348,Z 254.534,A -85,B 0,C 180,E1 -9315.661,E2 -9315.661} C_VEL
LIN {X 0,Y 432.364,Z 251.168,A -85,B 0,C 180,E1 -9318.392,E2 -9318.392} C_VEL
LIN {X 0,Y 432.301,Z 249.645,A -85,B 0,C 180,E1 -9319.824,E2 -9319.824} C_VEL
LIN {X 0,Y 432.302,Z 249.637,A -85,B 0,C 180,E1 -9323.023,E2 -9323.023} C_VEL
LIN {X 0,Y 432.347,Z 249.635,A -85,B 0,C 180,E1 -9325.997,E2 -9325.997} C_VEL
LIN {X 0,Y 432.382,Z 249.627,A -85,B 0,C 180,E1 -9329.745,E2 -9329.745} C_VEL
LIN {X 0,Y 432.387,Z 249.628,A -85,B 0,C 180,E1 -9333.373,E2 -9333.373} C_VEL
LIN {X 0,Y 432.362,Z 249.63,A -85,B 0,C 180,E1 -9336.024,E2 -9336.024} C_VEL
LIN {X 0,Y 432.366,Z 249.629,A -85,B 0,C 180,E1 -9339.048,E2 -9339.048} C_VEL
LIN {X 0,Y 432.367,Z 249.628,A -85,B 0,C 180,E1 -9342.012,E2 -9342.012} C_VEL
LIN {X 0,Y 432.389,Z 249.624,A -85,B 0,C 180,E1 -9344.928,E2 -9344.928} C_VEL
LIN {X 0,Y 432.448,Z 249.617,A -85,B 0,C 180,E1 -9347.804,E2 -9347.804} C_VEL
LIN {X 0,Y 432.482,Z 249.615,A -85,B 0,C 180,E1 -9351.591,E2 -9351.591} C_VEL
LIN {X 0,Y 432.581,Z 249.603,A -85,B 0,C 180,E1 -9354.407,E2 -9354.407} C_VEL
LIN {X 0,Y 432.597,Z 249.598,A -85,B 0,C 180,E1 -9358.139,E2 -9358.139} C_VEL
LIN {X 0,Y 432.72,Z 249.582,A -85,B 0,C 180,E1 -9360.001,E2 -9360.001} C_VEL
LIN {X 0,Y 432.597,Z 249.599,A -85,B 0,C 180,E1 -9362.795,E2 -9362.795} C_VEL
LIN {X 0,Y 432.559,Z 249.606,A -85,B 0,C 180,E1 -9366.532,E2 -9366.532} C_VEL
LIN {X 0,Y 432.435,Z 249.621,A -85,B 0,C 180,E1 -9369.354,E2 -9369.354} C_VEL
LIN {X 0,Y 432.423,Z 249.622,A -85,B 0,C 180,E1 -9372.805,E2 -9372.805} C_VEL
LIN {X 0,Y 432.406,Z 249.624,A -85,B 0,C 180,E1 -9376.48,E2 -9376.48} C_VEL
LIN {X 0,Y 432.332,Z 249.637,A -85,B 0,C 180,E1 -9379.962,E2 -9379.962} C_VEL
LIN {X 0,Y 432.313,Z 249.639,A -85,B 0,C 180,E1 -9382.966,E2 -9382.966} C_VEL
LIN {X 0,Y 432.34,Z 249.635,A -85,B 0,C 180,E1 -9385.003,E2 -9385.003} C_VEL
LIN {X 0,Y 432.342,Z 249.634,A -85,B 0,C 180,E1 -9388.127,E2 -9388.127} C_VEL
LIN {X 0,Y 432.316,Z 249.635,A -85,B 0,C 180,E1 -9391.347,E2 -9391.347} C_VEL
LIN {X 0,Y 432.336,Z 249.632,A -85,B 0,C 180,E1 -9394.678,E2 -9394.678} C_VEL
LIN {X 0,Y 432.334,Z 249.634,A -85,B 0,C 180,E1 -9398.151,E2 -9398.151} C_VEL
LIN {X 0,Y 432.33,Z 249.632,A -85,B 0,C 180,E1 -9401.603,E2 -9401.603} C_VEL
LIN {X 0,Y 432.332,Z 249.627,A -85,B 0,C 180,E1 -9404.349,E2 -9404.349} C_VEL
LIN {X 0,Y 432.302,Z 249.641,A -85,B 0,C 180,E1 -9407.019,E2 -9407.019} C_VEL
LIN {X 0,Y 432.333,Z 249.704,A -85,B 0,C 180,E1 -9408.721,E2 -9408.721} C_VEL
LIN {X 0,Y 433.028,Z 253.598,A -85,B 0,C 180,E1 -9411.173,E2 -9411.173} C_VEL
LIN {X 0,Y 433.492,Z 256.876,A -85,B 0,C 180,E1 -9413.141,E2 -9413.141} C_VEL
LIN {X 0,Y 433.632,Z 260.993,A -85,B 0,C 180,E1 -9415.442,E2 -9415.442} C_VEL
LIN {X 0,Y 433.151,Z 267.237,A -85,B 0,C 180,E1 -9418.722,E2 -9418.722} C_VEL
LIN {X 0,Y 432.795,Z 272.26,A -85,B 0,C 180,E1 -9421.27,E2 -9421.27} C_VEL
LIN {X 0,Y 432.355,Z 279.889,A -85,B 0,C 180,E1 -9425,E2 -9425} C_VEL
LIN {X 0,Y 432.014,Z 287.384,A -85,B 0,C 180,E1 -9428.53,E2 -9428.53} C_VEL
LIN {X 0,Y 431.694,Z 294.896,A -85,B 0,C 180,E1 -9431.982,E2 -9431.982} C_VEL
LIN {X 0,Y 431.67,Z 297.289,A -85,B 0,C 180,E1 -9433.067,E2 -9433.067} C_VEL
LIN {X 0,Y 434.434,Z 312.034,A -85,B 0,C 180,E1 -9433.654,E2 -9433.654} C_VEL
LIN {X 0,Y 435.806,Z 324.033,A -85,B 0,C 180,E1 -9434.269,E2 -9434.269} C_VEL
LIN {X 0,Y 435.045,Z 336.537,A -85,B 0,C 180,E1 -9435.021,E2 -9435.021} C_VEL
LIN {X 0,Y 434.258,Z 348.247,A -85,B 0,C 180,E1 -9435.951,E2 -9435.951} C_VEL
LIN {X 0,Y 433.62,Z 358.761,A -85,B 0,C 180,E1 -9437.004,E2 -9437.004} C_VEL
LIN {X 0,Y 433.099,Z 367.374,A -85,B 0,C 180,E1 -9438.06,E2 -9438.06} C_VEL
LIN {X 0,Y 432.414,Z 375.331,A -85,B 0,C 180,E1 -9439.228,E2 -9439.228} C_VEL
LIN {X 0,Y 431.979,Z 383.146,A -85,B 0,C 180,E1 -9440.637,E2 -9440.637} C_VEL
LIN {X 0,Y 431.615,Z 389.407,A -85,B 0,C 180,E1 -9442.045,E2 -9442.045} C_VEL
LIN {X 0,Y 431.359,Z 395.005,A -85,B 0,C 180,E1 -9443.65,E2 -9443.65} C_VEL
LIN {X 0,Y 431.271,Z 399.345,A -85,B 0,C 180,E1 -9445.327,E2 -9445.327} C_VEL
LIN {X 0,Y 431.187,Z 401.126,A -85,B 0,C 180,E1 -9446.262,E2 -9446.262} C_VEL
LIN {X 0,Y 431.236,Z 402.48,A -85,B 0,C 180,E1 -9447.198,E2 -9447.198} C_VEL
LIN {X 0,Y 431.204,Z 403.44,A -85,B 0,C 180,E1 -9448.132,E2 -9448.132} C_VEL
LIN {X 0,Y 431.17,Z 404.012,A -85,B 0,C 180,E1 -9449.066,E2 -9449.066} C_VEL
LIN {X 0,Y 431.168,Z 404.16,A -85,B 0,C 180,E1 -9450,E2 -9450} C_VEL
LIN {X 0,Y 431.204,Z 403.258,A -85,B 0,C 180,E1 -9451.868,E2 -9451.868} C_VEL
LIN {X 0,Y 431.237,Z 402.225,A -85,B 0,C 180,E1 -9452.802,E2 -9452.802} C_VEL
LIN {X 0,Y 431.188,Z 400.75,A -85,B 0,C 180,E1 -9453.738,E2 -9453.738} C_VEL
LIN {X 0,Y 431.296,Z 397.737,A -85,B 0,C 180,E1 -9455.142,E2 -9455.142} C_VEL
LIN {X 0,Y 431.379,Z 393.659,A -85,B 0,C 180,E1 -9456.548,E2 -9456.548} C_VEL
LIN {X 0,Y 431.621,Z 387.39,A -85,B 0,C 180,E1 -9458.191,E2 -9458.191} C_VEL
LIN {X 0,Y 431.992,Z 380.56,A -85,B 0,C 180,E1 -9459.599,E2 -9459.599} C_VEL
LIN {X 0,Y 432.443,Z 372.045,A -85,B 0,C 180,E1 -9461.009,E2 -9461.009} C_VEL
LIN {X 0,Y 433.02,Z 363.277,A -85,B 0,C 180,E1 -9462.18,E2 -9462.18} C_VEL
LIN {X 0,Y 433.63,Z 352.824,A -85,B 0,C 180,E1 -9463.318,E2 -9463.318} C_VEL
LIN {X 0,Y 434.241,Z 341.688,A -85,B 0,C 180,E1 -9464.289,E2 -9464.289} C_VEL
LIN {X 0,Y 434.937,Z 329.58,A -85,B 0,C 180,E1 -9465.103,E2 -9465.103} C_VEL
LIN {X 0,Y 435.156,Z 322.03,A -85,B 0,C 180,E1 -9465.515,E2 -9465.515} C_VEL
LIN {X 0,Y 433.422,Z 309.348,A -85,B 0,C 180,E1 -9466.105,E2 -9466.105} C_VEL
LIN {X 0,Y 431.543,Z 297.498,A -85,B 0,C 180,E1 -9466.507,E2 -9466.507} C_VEL
LIN {X 0,Y 431.744,Z 291.339,A -85,B 0,C 180,E1 -9469.241,E2 -9469.241} C_VEL
LIN {X 0,Y 431.982,Z 285.256,A -85,B 0,C 180,E1 -9471.974,E2 -9471.974} C_VEL
LIN {X 0,Y 432.27,Z 277.494,A -85,B 0,C 180,E1 -9475.521,E2 -9475.521} C_VEL
LIN {X 0,Y 432.644,Z 269.749,A -85,B 0,C 180,E1 -9479.164,E2 -9479.164} C_VEL
LIN {X 0,Y 433.048,Z 262.962,A -85,B 0,C 180,E1 -9482.443,E2 -9482.443} C_VEL
LIN {X 0,Y 433.312,Z 257.532,A -85,B 0,C 180,E1 -9485.154,E2 -9485.154} C_VEL
LIN {X 0,Y 432.989,Z 253.421,A -85,B 0,C 180,E1 -9487.312,E2 -9487.312} C_VEL
LIN {X 0,Y 432.374,Z 249.63,A -85,B 0,C 180,E1 -9489.489,E2 -9489.489} C_VEL
LIN {X 0,Y 432.298,Z 249.638,A -85,B 0,C 180,E1 -9493.062,E2 -9493.062} C_VEL
LIN {X 0,Y 432.308,Z 249.632,A -85,B 0,C 180,E1 -9495.667,E2 -9495.667} C_VEL
LIN {X 0,Y 432.303,Z 249.635,A -85,B 0,C 180,E1 -9498.401,E2 -9498.401} C_VEL
LIN {X 0,Y 432.317,Z 249.632,A -85,B 0,C 180,E1 -9501.847,E2 -9501.847} C_VEL
LIN {X 0,Y 432.321,Z 249.632,A -85,B 0,C 180,E1 -9505.32,E2 -9505.32} C_VEL
LIN {X 0,Y 432.316,Z 249.635,A -85,B 0,C 180,E1 -9508.653,E2 -9508.653} C_VEL
LIN {X 0,Y 432.331,Z 249.632,A -85,B 0,C 180,E1 -9511.872,E2 -9511.872} C_VEL
LIN {X 0,Y 432.372,Z 249.626,A -85,B 0,C 180,E1 -9515.538,E2 -9515.538} C_VEL
LIN {X 0,Y 432.344,Z 249.63,A -85,B 0,C 180,E1 -9519.045,E2 -9519.045} C_VEL
LIN {X 0,Y 432.367,Z 249.63,A -85,B 0,C 180,E1 -9522.01,E2 -9522.01} C_VEL
LIN {X 0,Y 432.388,Z 249.625,A -85,B 0,C 180,E1 -9524.925,E2 -9524.925} C_VEL
LIN {X 0,Y 432.452,Z 249.619,A -85,B 0,C 180,E1 -9527.802,E2 -9527.802} C_VEL
LIN {X 0,Y 432.484,Z 249.614,A -85,B 0,C 180,E1 -9531.589,E2 -9531.589} C_VEL
LIN {X 0,Y 432.588,Z 249.601,A -85,B 0,C 180,E1 -9534.405,E2 -9534.405} C_VEL
LIN {X 0,Y 432.596,Z 249.599,A -85,B 0,C 180,E1 -9538.137,E2 -9538.137} C_VEL
LIN {X 0,Y 432.725,Z 249.583,A -85,B 0,C 180,E1 -9539.999,E2 -9539.999} C_VEL
LIN {X 0,Y 432.597,Z 249.598,A -85,B 0,C 180,E1 -9542.792,E2 -9542.792} C_VEL
LIN {X 0,Y 432.564,Z 249.603,A -85,B 0,C 180,E1 -9546.529,E2 -9546.529} C_VEL
LIN {X 0,Y 432.434,Z 249.619,A -85,B 0,C 180,E1 -9549.352,E2 -9549.352} C_VEL
LIN {X 0,Y 432.42,Z 249.62,A -85,B 0,C 180,E1 -9552.803,E2 -9552.803} C_VEL
LIN {X 0,Y 432.401,Z 249.622,A -85,B 0,C 180,E1 -9556.478,E2 -9556.478} C_VEL
LIN {X 0,Y 432.327,Z 249.633,A -85,B 0,C 180,E1 -9559.96,E2 -9559.96} C_VEL
LIN {X 0,Y 432.308,Z 249.634,A -85,B 0,C 180,E1 -9562.963,E2 -9562.963} C_VEL
LIN {X 0,Y 432.353,Z 249.628,A -85,B 0,C 180,E1 -9566.032,E2 -9566.032} C_VEL
LIN {X 0,Y 432.34,Z 249.632,A -85,B 0,C 180,E1 -9569.186,E2 -9569.186} C_VEL
LIN {X 0,Y 432.313,Z 249.632,A -85,B 0,C 180,E1 -9572.293,E2 -9572.293} C_VEL
LIN {X 0,Y 432.329,Z 249.631,A -85,B 0,C 180,E1 -9574.676,E2 -9574.676} C_VEL
LIN {X 0,Y 432.341,Z 249.628,A -85,B 0,C 180,E1 -9578.148,E2 -9578.148} C_VEL
LIN {X 0,Y 432.361,Z 249.625,A -85,B 0,C 180,E1 -9581.608,E2 -9581.608} C_VEL
LIN {X 0,Y 432.366,Z 249.625,A -85,B 0,C 180,E1 -9584.341,E2 -9584.341} C_VEL
LIN {X 0,Y 432.322,Z 249.631,A -85,B 0,C 180,E1 -9588.203,E2 -9588.203} C_VEL
LIN {X 0,Y 432.338,Z 249.629,A -85,B 0,C 180,E1 -9591.284,E2 -9591.284} C_VEL
LIN {X 0,Y 432.333,Z 249.633,A -85,B 0,C 180,E1 -9594.368,E2 -9594.368} C_VEL
LIN {X 0,Y 432.31,Z 249.632,A -85,B 0,C 180,E1 -9597.557,E2 -9597.557} C_VEL
LIN {X 0,Y 432.33,Z 249.631,A -85,B 0,C 180,E1 -9600.812,E2 -9600.812} C_VEL
LIN {X 0,Y 432.338,Z 249.632,A -85,B 0,C 180,E1 -9603.966,E2 -9603.966} C_VEL
LIN {X 0,Y 432.319,Z 249.635,A -85,B 0,C 180,E1 -9606.021,E2 -9606.021} C_VEL
LIN {X 0,Y 432.156,Z 249.656,A -85,B 0,C 180,E1 -9608.035,E2 -9608.035} C_VEL
LIN {X 0,Y 432.136,Z 252.83,A -85,B 0,C 180,E1 -9610.604,E2 -9610.604} C_VEL
LIN {X 0,Y 431.981,Z 257.42,A -85,B 0,C 180,E1 -9613.944,E2 -9613.944} C_VEL
LIN {X 0,Y 431.915,Z 262.809,A -85,B 0,C 180,E1 -9617.788,E2 -9617.788} C_VEL
LIN {X 0,Y 431.735,Z 268.254,A -85,B 0,C 180,E1 -9621.576,E2 -9621.576} C_VEL
LIN {X 0,Y 431.764,Z 270.98,A -85,B 0,C 180,E1 -9623.458,E2 -9623.458} C_VEL
LIN {X 0,Y 431.64,Z 275.612,A -85,B 0,C 180,E1 -9626.587,E2 -9626.587} C_VEL
LIN {X 0,Y 434.199,Z 289.416,A -85,B 0,C 180,E1 -9627.115,E2 -9627.115} C_VEL
LIN {X 0,Y 435.55,Z 297.518,A -85,B 0,C 180,E1 -9627.515,E2 -9627.515} C_VEL
LIN {X 0,Y 435.037,Z 308.896,A -85,B 0,C 180,E1 -9628.148,E2 -9628.148} C_VEL
LIN {X 0,Y 434.438,Z 320.096,A -85,B 0,C 180,E1 -9628.957,E2 -9628.957} C_VEL
LIN {X 0,Y 433.828,Z 330.952,A -85,B 0,C 180,E1 -9629.947,E2 -9629.947} C_VEL
LIN {X 0,Y 432.977,Z 335.592,A -85,B 0,C 180,E1 -9630.419,E2 -9630.419} C_VEL
LIN {X 0,Y 429.659,Z 342.802,A -85,B 0,C 180,E1 -9631.213,E2 -9631.213} C_VEL
LIN {X 0,Y 426.283,Z 349.435,A -85,B 0,C 180,E1 -9632.097,E2 -9632.097} C_VEL
LIN {X 0,Y 425.354,Z 353.17,A -85,B 0,C 180,E1 -9632.702,E2 -9632.702} C_VEL
LIN {X 0,Y 424.906,Z 361.271,A -85,B 0,C 180,E1 -9634.268,E2 -9634.268} C_VEL
LIN {X 0,Y 424.611,Z 367.143,A -85,B 0,C 180,E1 -9635.699,E2 -9635.699} C_VEL
LIN {X 0,Y 424.411,Z 371.781,A -85,B 0,C 180,E1 -9637.134,E2 -9637.134} C_VEL
LIN {X 0,Y 424.198,Z 375.326,A -85,B 0,C 180,E1 -9638.575,E2 -9638.575} C_VEL
LIN {X 0,Y 424.092,Z 377.119,A -85,B 0,C 180,E1 -9639.539,E2 -9639.539} C_VEL
LIN {X 0,Y 424.064,Z 378.47,A -85,B 0,C 180,E1 -9640.504,E2 -9640.504} C_VEL
LIN {X 0,Y 424.076,Z 379.815,A -85,B 0,C 180,E1 -9642.11,E2 -9642.11} C_VEL
LIN {X 0,Y 423.971,Z 380.084,A -85,B 0,C 180,E1 -9643.419,E2 -9643.419} C_VEL
LIN {X 0,Y 423.969,Z 379.786,A -85,B 0,C 180,E1 -9644.397,E2 -9644.397} C_VEL
LIN {X 0,Y 424.11,Z 378.362,A -85,B 0,C 180,E1 -9646.034,E2 -9646.034} C_VEL
LIN {X 0,Y 424.253,Z 375.395,A -85,B 0,C 180,E1 -9647.846,E2 -9647.846} C_VEL
LIN {X 0,Y 424.488,Z 371.753,A -85,B 0,C 180,E1 -9649.337,E2 -9649.337} C_VEL
LIN {X 0,Y 424.79,Z 366.896,A -85,B 0,C 180,E1 -9650.836,E2 -9650.836} C_VEL
LIN {X 0,Y 425.246,Z 360.665,A -85,B 0,C 180,E1 -9652.34,E2 -9652.34} C_VEL
LIN {X 0,Y 425.848,Z 352.819,A -85,B 0,C 180,E1 -9653.849,E2 -9653.849} C_VEL
LIN {X 0,Y 426.482,Z 344.693,A -85,B 0,C 180,E1 -9655.106,E2 -9655.106} C_VEL
LIN {X 0,Y 427.209,Z 334.593,A -85,B 0,C 180,E1 -9656.37,E2 -9656.37} C_VEL
LIN {X 0,Y 428.009,Z 324.025,A -85,B 0,C 180,E1 -9657.432,E2 -9657.432} C_VEL
LIN {X 0,Y 428.627,Z 313.732,A -85,B 0,C 180,E1 -9658.265,E2 -9658.265} C_VEL
LIN {X 0,Y 429.369,Z 302.038,A -85,B 0,C 180,E1 -9658.997,E2 -9658.997} C_VEL
LIN {X 0,Y 429.42,Z 298.378,A -85,B 0,C 180,E1 -9659.196,E2 -9659.196} C_VEL
LIN {X 0,Y 427.078,Z 286.348,A -85,B 0,C 180,E1 -9659.839,E2 -9659.839} C_VEL
LIN {X 0,Y 424.453,Z 275.973,A -85,B 0,C 180,E1 -9660.317,E2 -9660.317} C_VEL
LIN {X 0,Y 424.556,Z 272.058,A -85,B 0,C 180,E1 -9663.111,E2 -9663.111} C_VEL
LIN {X 0,Y 424.691,Z 267.338,A -85,B 0,C 180,E1 -9666.565,E2 -9666.565} C_VEL
LIN {X 0,Y 424.871,Z 264.108,A -85,B 0,C 180,E1 -9668.975,E2 -9668.975} C_VEL
LIN {X 0,Y 425.046,Z 259.284,A -85,B 0,C 180,E1 -9672.68,E2 -9672.68} C_VEL
LIN {X 0,Y 425.32,Z 255.044,A -85,B 0,C 180,E1 -9676.054,E2 -9676.054} C_VEL
LIN {X 0,Y 425.342,Z 251.916,A -85,B 0,C 180,E1 -9678.631,E2 -9678.631} C_VEL
LIN {X 0,Y 425.253,Z 250.523,A -85,B 0,C 180,E1 -9679.871,E2 -9679.871} C_VEL
LIN {X 0,Y 425.27,Z 250.515,A -85,B 0,C 180,E1 -9682.488,E2 -9682.488} C_VEL
LIN {X 0,Y 425.295,Z 250.513,A -85,B 0,C 180,E1 -9685.818,E2 -9685.818} C_VEL
LIN {X 0,Y 425.288,Z 250.511,A -85,B 0,C 180,E1 -9689.237,E2 -9689.237} C_VEL
LIN {X 0,Y 425.337,Z 250.503,A -85,B 0,C 180,E1 -9692.443,E2 -9692.443} C_VEL
LIN {X 0,Y 425.34,Z 250.503,A -85,B 0,C 180,E1 -9695.603,E2 -9695.603} C_VEL
LIN {X 0,Y 425.309,Z 250.507,A -85,B 0,C 180,E1 -9698.684,E2 -9698.684} C_VEL
LIN {X 0,Y 425.322,Z 250.504,A -85,B 0,C 180,E1 -9701.704,E2 -9701.704} C_VEL
LIN {X 0,Y 425.344,Z 250.501,A -85,B 0,C 180,E1 -9704.672,E2 -9704.672} C_VEL
LIN {X 0,Y 425.401,Z 250.495,A -85,B 0,C 180,E1 -9707.599,E2 -9707.599} C_VEL
LIN {X 0,Y 425.432,Z 250.494,A -85,B 0,C 180,E1 -9711.451,E2 -9711.451} C_VEL
LIN {X 0,Y 425.538,Z 250.48,A -85,B 0,C 180,E1 -9714.314,E2 -9714.314} C_VEL
LIN {X 0,Y 425.567,Z 250.474,A -85,B 0,C 180,E1 -9718.108,E2 -9718.108} C_VEL
LIN {X 0,Y 425.69,Z 250.458,A -85,B 0,C 180,E1 -9720.001,E2 -9720.001} C_VEL
LIN {X 0,Y 425.549,Z 250.477,A -85,B 0,C 180,E1 -9722.841,E2 -9722.841} C_VEL
LIN {X 0,Y 425.518,Z 250.483,A -85,B 0,C 180,E1 -9726.64,E2 -9726.64} C_VEL
LIN {X 0,Y 425.393,Z 250.499,A -85,B 0,C 180,E1 -9729.511,E2 -9729.511} C_VEL
LIN {X 0,Y 425.386,Z 250.498,A -85,B 0,C 180,E1 -9732.905,E2 -9732.905} C_VEL
LIN {X 0,Y 425.355,Z 250.503,A -85,B 0,C 180,E1 -9736.606,E2 -9736.606} C_VEL
LIN {X 0,Y 425.322,Z 250.507,A -85,B 0,C 180,E1 -9739.637,E2 -9739.637} C_VEL
LIN {X 0,Y 425.301,Z 250.513,A -85,B 0,C 180,E1 -9743.366,E2 -9743.366} C_VEL
LIN {X 0,Y 425.323,Z 250.51,A -85,B 0,C 180,E1 -9746.498,E2 -9746.498} C_VEL
LIN {X 0,Y 425.281,Z 250.513,A -85,B 0,C 180,E1 -9749.721,E2 -9749.721} C_VEL
LIN {X 0,Y 425.278,Z 250.512,A -85,B 0,C 180,E1 -9753.049,E2 -9753.049} C_VEL
LIN {X 0,Y 425.278,Z 250.511,A -85,B 0,C 180,E1 -9755.93,E2 -9755.93} C_VEL
LIN {X 0,Y 425.292,Z 250.508,A -85,B 0,C 180,E1 -9759.044,E2 -9759.044} C_VEL
LIN {X 0,Y 425.273,Z 250.511,A -85,B 0,C 180,E1 -9762.654,E2 -9762.654} C_VEL
LIN {X 0,Y 425.256,Z 250.518,A -85,B 0,C 180,E1 -9766.045,E2 -9766.045} C_VEL
LIN {X 0,Y 425.286,Z 250.518,A -85,B 0,C 180,E1 -9768.337,E2 -9768.337} C_VEL
LIN {X 0,Y 426.059,Z 254.933,A -85,B 0,C 180,E1 -9771.185,E2 -9771.185} C_VEL
LIN {X 0,Y 426.578,Z 259.345,A -85,B 0,C 180,E1 -9773.833,E2 -9773.833} C_VEL
LIN {X 0,Y 426.532,Z 263.094,A -85,B 0,C 180,E1 -9775.93,E2 -9775.93} C_VEL
LIN {X 0,Y 426.077,Z 269.32,A -85,B 0,C 180,E1 -9779.248,E2 -9779.248} C_VEL
LIN {X 0,Y 425.554,Z 275.615,A -85,B 0,C 180,E1 -9782.458,E2 -9782.458} C_VEL
LIN {X 0,Y 425.23,Z 281.971,A -85,B 0,C 180,E1 -9785.595,E2 -9785.595} C_VEL
LIN {X 0,Y 424.934,Z 288.372,A -85,B 0,C 180,E1 -9788.663,E2 -9788.663} C_VEL
LIN {X 0,Y 424.629,Z 295.864,A -85,B 0,C 180,E1 -9792.171,E2 -9792.171} C_VEL
LIN {X 0,Y 424.611,Z 297.336,A -85,B 0,C 180,E1 -9792.754,E2 -9792.754} C_VEL
LIN {X 0,Y 427.236,Z 310.419,A -85,B 0,C 180,E1 -9793.272,E2 -9793.272} C_VEL
LIN {X 0,Y 428.814,Z 322.322,A -85,B 0,C 180,E1 -9793.884,E2 -9793.884} C_VEL
LIN {X 0,Y 428.749,Z 329.676,A -85,B 0,C 180,E1 -9794.308,E2 -9794.308} C_VEL
LIN {X 0,Y 428.009,Z 340.004,A -85,B 0,C 180,E1 -9795.012,E2 -9795.012} C_VEL
LIN {X 0,Y 427.193,Z 350.991,A -85,B 0,C 180,E1 -9795.954,E2 -9795.954} C_VEL
LIN {X 0,Y 426.489,Z 361.914,A -85,B 0,C 180,E1 -9797.147,E2 -9797.147} C_VEL
LIN {X 0,Y 425.827,Z 370.778,A -85,B 0,C 180,E1 -9798.336,E2 -9798.336} C_VEL
LIN {X 0,Y 425.194,Z 379.454,A -85,B 0,C 180,E1 -9799.765,E2 -9799.765} C_VEL
LIN {X 0,Y 424.733,Z 386.391,A -85,B 0,C 180,E1 -9801.196,E2 -9801.196} C_VEL
LIN {X 0,Y 424.406,Z 392.774,A -85,B 0,C 180,E1 -9802.866,E2 -9802.866} C_VEL
LIN {X 0,Y 424.195,Z 396.977,A -85,B 0,C 180,E1 -9804.295,E2 -9804.295} C_VEL
LIN {X 0,Y 424.201,Z 399.215,A -85,B 0,C 180,E1 -9805.248,E2 -9805.248} C_VEL
LIN {X 0,Y 424.099,Z 400.974,A -85,B 0,C 180,E1 -9806.199,E2 -9806.199} C_VEL
LIN {X 0,Y 424.132,Z 402.317,A -85,B 0,C 180,E1 -9807.151,E2 -9807.151} C_VEL
LIN {X 0,Y 424.13,Z 403.267,A -85,B 0,C 180,E1 -9808.101,E2 -9808.101} C_VEL
LIN {X 0,Y 424.089,Z 403.826,A -85,B 0,C 180,E1 -9809.051,E2 -9809.051} C_VEL
LIN {X 0,Y 424.085,Z 403.954,A -85,B 0,C 180,E1 -9810,E2 -9810} C_VEL
LIN {X 0,Y 424.13,Z 403.032,A -85,B 0,C 180,E1 -9811.899,E2 -9811.899} C_VEL
LIN {X 0,Y 424.134,Z 401.987,A -85,B 0,C 180,E1 -9812.849,E2 -9812.849} C_VEL
LIN {X 0,Y 424.1,Z 400.49,A -85,B 0,C 180,E1 -9813.801,E2 -9813.801} C_VEL
LIN {X 0,Y 424.208,Z 397.452,A -85,B 0,C 180,E1 -9815.228,E2 -9815.228} C_VEL
LIN {X 0,Y 424.302,Z 393.348,A -85,B 0,C 180,E1 -9816.658,E2 -9816.658} C_VEL
LIN {X 0,Y 424.552,Z 387.049,A -85,B 0,C 180,E1 -9818.328,E2 -9818.328} C_VEL
LIN {X 0,Y 424.945,Z 380.186,A -85,B 0,C 180,E1 -9819.76,E2 -9819.76} C_VEL
LIN {X 0,Y 425.324,Z 373.171,A -85,B 0,C 180,E1 -9820.954,E2 -9820.954} C_VEL
LIN {X 0,Y 425.931,Z 364.727,A -85,B 0,C 180,E1 -9822.144,E2 -9822.144} C_VEL
LIN {X 0,Y 426.486,Z 355.466,A -85,B 0,C 180,E1 -9823.217,E2 -9823.217} C_VEL
LIN {X 0,Y 427.158,Z 343.944,A -85,B 0,C 180,E1 -9824.288,E2 -9824.288} C_VEL
LIN {X 0,Y 427.817,Z 332.626,A -85,B 0,C 180,E1 -9825.116,E2 -9825.116} C_VEL
LIN {X 0,Y 428.185,Z 322.467,A -85,B 0,C 180,E1 -9825.701,E2 -9825.701} C_VEL
LIN {X 0,Y 426.44,Z 309.513,A -85,B 0,C 180,E1 -9826.324,E2 -9826.324} C_VEL
LIN {X 0,Y 424.492,Z 297.287,A -85,B 0,C 180,E1 -9826.755,E2 -9826.755} C_VEL
LIN {X 0,Y 424.684,Z 290.509,A -85,B 0,C 180,E1 -9829.83,E2 -9829.83} C_VEL
LIN {X 0,Y 424.944,Z 283.879,A -85,B 0,C 180,E1 -9832.871,E2 -9832.871} C_VEL
LIN {X 0,Y 425.277,Z 277.256,A -85,B 0,C 180,E1 -9835.971,E2 -9835.971} C_VEL
LIN {X 0,Y 425.648,Z 269.496,A -85,B 0,C 180,E1 -9839.691,E2 -9839.691} C_VEL
LIN {X 0,Y 426.047,Z 262.841,A -85,B 0,C 180,E1 -9842.98,E2 -9842.98} C_VEL
LIN {X 0,Y 426.303,Z 258.399,A -85,B 0,C 180,E1 -9845.239,E2 -9845.239} C_VEL
LIN {X 0,Y 425.881,Z 253.944,A -85,B 0,C 180,E1 -9847.631,E2 -9847.631} C_VEL
LIN {X 0,Y 425.347,Z 250.505,A -85,B 0,C 180,E1 -9849.556,E2 -9849.556} C_VEL
LIN {X 0,Y 425.242,Z 250.514,A -85,B 0,C 180,E1 -9853.348,E2 -9853.348} C_VEL
LIN {X 0,Y 425.232,Z 250.514,A -85,B 0,C 180,E1 -9856.039,E2 -9856.039} C_VEL
LIN {X 0,Y 425.239,Z 250.513,A -85,B 0,C 180,E1 -9859.485,E2 -9859.485} C_VEL
LIN {X 0,Y 425.265,Z 250.514,A -85,B 0,C 180,E1 -9862.489,E2 -9862.489} C_VEL
LIN {X 0,Y 425.281,Z 250.508,A -85,B 0,C 180,E1 -9865.814,E2 -9865.814} C_VEL
LIN {X 0,Y 425.286,Z 250.509,A -85,B 0,C 180,E1 -9869.238,E2 -9869.238} C_VEL
LIN {X 0,Y 425.256,Z 250.515,A -85,B 0,C 180,E1 -9872.435,E2 -9872.435} C_VEL
LIN {X 0,Y 425.34,Z 250.502,A -85,B 0,C 180,E1 -9875.6,E2 -9875.6} C_VEL
LIN {X 0,Y 425.287,Z 250.509,A -85,B 0,C 180,E1 -9878.68,E2 -9878.68} C_VEL
LIN {X 0,Y 425.323,Z 250.505,A -85,B 0,C 180,E1 -9881.701,E2 -9881.701} C_VEL
LIN {X 0,Y 425.341,Z 250.503,A -85,B 0,C 180,E1 -9884.669,E2 -9884.669} C_VEL
LIN {X 0,Y 425.405,Z 250.495,A -85,B 0,C 180,E1 -9887.597,E2 -9887.597} C_VEL
LIN {X 0,Y 425.435,Z 250.491,A -85,B 0,C 180,E1 -9891.449,E2 -9891.449} C_VEL
LIN {X 0,Y 425.545,Z 250.478,A -85,B 0,C 180,E1 -9894.312,E2 -9894.312} C_VEL
LIN {X 0,Y 425.566,Z 250.475,A -85,B 0,C 180,E1 -9898.106,E2 -9898.106} C_VEL
LIN {X 0,Y 425.695,Z 250.459,A -85,B 0,C 180,E1 -9899.999,E2 -9899.999} C_VEL
LIN {X 0,Y 425.549,Z 250.476,A -85,B 0,C 180,E1 -9902.839,E2 -9902.839} C_VEL
LIN {X 0,Y 425.521,Z 250.479,A -85,B 0,C 180,E1 -9906.655,E2 -9906.655} C_VEL
LIN {X 0,Y 425.392,Z 250.496,A -85,B 0,C 180,E1 -9909.508,E2 -9909.508} C_VEL
LIN {X 0,Y 425.383,Z 250.497,A -85,B 0,C 180,E1 -9912.903,E2 -9912.903} C_VEL
LIN {X 0,Y 425.35,Z 250.5,A -85,B 0,C 180,E1 -9916.604,E2 -9916.604} C_VEL
LIN {X 0,Y 425.317,Z 250.508,A -85,B 0,C 180,E1 -9919.635,E2 -9919.635} C_VEL
LIN {X 0,Y 425.296,Z 250.51,A -85,B 0,C 180,E1 -9923.364,E2 -9923.364} C_VEL
LIN {X 0,Y 425.337,Z 250.502,A -85,B 0,C 180,E1 -9926.844,E2 -9926.844} C_VEL
LIN {X 0,Y 425.306,Z 250.506,A -85,B 0,C 180,E1 -9929.717,E2 -9929.717} C_VEL
LIN {X 0,Y 425.27,Z 250.513,A -85,B 0,C 180,E1 -9933.047,E2 -9933.047} C_VEL
LIN {X 0,Y 425.273,Z 250.508,A -85,B 0,C 180,E1 -9935.929,E2 -9935.929} C_VEL
LIN {X 0,Y 425.302,Z 250.511,A -85,B 0,C 180,E1 -9939.046,E2 -9939.046} C_VEL
LIN {X 0,Y 425.319,Z 250.506,A -85,B 0,C 180,E1 -9942.645,E2 -9942.645} C_VEL
LIN {X 0,Y 425.256,Z 250.51,A -85,B 0,C 180,E1 -9946.045,E2 -9946.045} C_VEL
LIN {X 0,Y 425.263,Z 250.514,A -85,B 0,C 180,E1 -9948.621,E2 -9948.621} C_VEL
LIN {X 0,Y 425.3,Z 250.506,A -85,B 0,C 180,E1 -9951.103,E2 -9951.103} C_VEL
LIN {X 0,Y 425.288,Z 250.511,A -85,B 0,C 180,E1 -9954.664,E2 -9954.664} C_VEL
LIN {X 0,Y 425.252,Z 250.513,A -85,B 0,C 180,E1 -9958.073,E2 -9958.073} C_VEL
LIN {X 0,Y 425.318,Z 250.503,A -85,B 0,C 180,E1 -9961.368,E2 -9961.368} C_VEL
LIN {X 0,Y 425.333,Z 250.502,A -85,B 0,C 180,E1 -9963.505,E2 -9963.505} C_VEL
LIN {X 0,Y 425.227,Z 250.516,A -85,B 0,C 180,E1 -9966.631,E2 -9966.631} C_VEL
LIN {X 0,Y 425.147,Z 250.527,A -85,B 0,C 180,E1 -9967.773,E2 -9967.773} C_VEL
LIN {X 0,Y 425.061,Z 251.086,A -85,B 0,C 180,E1 -9968.67,E2 -9968.67} C_VEL
LIN {X 0,Y 425.024,Z 255.109,A -85,B 0,C 180,E1 -9971.689,E2 -9971.689} C_VEL
LIN {X 0,Y 424.875,Z 259.141,A -85,B 0,C 180,E1 -9974.654,E2 -9974.654} C_VEL
LIN {X 0,Y 424.868,Z 263.211,A -85,B 0,C 180,E1 -9977.582,E2 -9977.582} C_VEL
LIN {X 0,Y 424.679,Z 268.667,A -85,B 0,C 180,E1 -9981.435,E2 -9981.435} C_VEL
LIN {X 0,Y 424.704,Z 271.42,A -85,B 0,C 180,E1 -9983.348,E2 -9983.348} C_VEL
LIN {X 0,Y 424.557,Z 275.809,A -85,B 0,C 180,E1 -9986.352,E2 -9986.352} C_VEL
LIN {X 0,Y 427.025,Z 289.101,A -85,B 0,C 180,E1 -9986.86,E2 -9986.86} C_VEL
LIN {X 0,Y 428.638,Z 297.745,A -85,B 0,C 180,E1 -9987.298,E2 -9987.298} C_VEL
LIN {X 0,Y 428.081,Z 309.984,A -85,B 0,C 180,E1 -9988.001,E2 -9988.001} C_VEL
LIN {X 0,Y 427.355,Z 322.437,A -85,B 0,C 180,E1 -9988.94,E2 -9988.94} C_VEL
LIN {X 0,Y 426.739,Z 333.34,A -85,B 0,C 180,E1 -9990,E2 -9990} C_VEL
LIN {X 0,Y 426.073,Z 343.121,A -85,B 0,C 180,E1 -9991.181,E2 -9991.181} C_VEL
LIN {X 0,Y 425.506,Z 351.151,A -85,B 0,C 180,E1 -9992.366,E2 -9992.366} C_VEL
LIN {X 0,Y 425.354,Z 353.17,A -85,B 0,C 180,E1 -9992.702,E2 -9992.702} C_VEL
LIN {X 0,Y 424.485,Z 356.749,A -85,B 0,C 180,E1 -9993.332,E2 -9993.332} C_VEL
LIN {X 0,Y 421.343,Z 362.133,A -85,B 0,C 180,E1 -9994.379,E2 -9994.379} C_VEL
LIN {X 0,Y 418.246,Z 366.842,A -85,B 0,C 180,E1 -9995.49,E2 -9995.49} C_VEL
LIN {X 0,Y 417.455,Z 369.368,A -85,B 0,C 180,E1 -9996.211,E2 -9996.211} C_VEL
LIN {X 0,Y 417.264,Z 373.727,A -85,B 0,C 180,E1 -9997.744,E2 -9997.744} C_VEL
LIN {X 0,Y 417.097,Z 375.897,A -85,B 0,C 180,E1 -9998.722,E2 -9998.722} C_VEL
LIN {X 0,Y 416.983,Z 377.597,A -85,B 0,C 180,E1 -9999.703,E2 -9999.703} C_VEL
LIN {X 0,Y 416.984,Z 378.884,A -85,B 0,C 180,E1 -10000.684,E2 -10000.684} C_VEL
LIN {X 0,Y 416.986,Z 380.035,A -85,B 0,C 180,E1 -10002.172,E2 -10002.172} C_VEL
LIN {X 0,Y 416.876,Z 380.255,A -85,B 0,C 180,E1 -10003.652,E2 -10003.652} C_VEL
LIN {X 0,Y 416.895,Z 379.895,A -85,B 0,C 180,E1 -10004.647,E2 -10004.647} C_VEL
LIN {X 0,Y 417.026,Z 378.541,A -85,B 0,C 180,E1 -10006.143,E2 -10006.143} C_VEL
LIN {X 0,Y 417.241,Z 375.181,A -85,B 0,C 180,E1 -10008.156,E2 -10008.156} C_VEL
LIN {X 0,Y 417.475,Z 371.395,A -85,B 0,C 180,E1 -10009.675,E2 -10009.675} C_VEL
LIN {X 0,Y 417.829,Z 366.384,A -85,B 0,C 180,E1 -10011.2,E2 -10011.2} C_VEL
LIN {X 0,Y 418.351,Z 359.985,A -85,B 0,C 180,E1 -10012.729,E2 -10012.729} C_VEL
LIN {X 0,Y 418.877,Z 353.361,A -85,B 0,C 180,E1 -10014.008,E2 -10014.008} C_VEL
LIN {X 0,Y 419.499,Z 345.745,A -85,B 0,C 180,E1 -10015.224,E2 -10015.224} C_VEL
LIN {X 0,Y 420.224,Z 336.471,A -85,B 0,C 180,E1 -10016.441,E2 -10016.441} C_VEL
LIN {X 0,Y 421.103,Z 325.533,A -85,B 0,C 180,E1 -10017.589,E2 -10017.589} C_VEL
LIN {X 0,Y 421.763,Z 315.382,A -85,B 0,C 180,E1 -10018.447,E2 -10018.447} C_VEL
LIN {X 0,Y 422.533,Z 304.497,A -85,B 0,C 180,E1 -10019.172,E2 -10019.172} C_VEL
LIN {X 0,Y 422.541,Z 298.682,A -85,B 0,C 180,E1 -10019.506,E2 -10019.506} C_VEL
LIN {X 0,Y 420.141,Z 286.829,A -85,B 0,C 180,E1 -10020.163,E2 -10020.163} C_VEL
LIN {X 0,Y 417.396,Z 276.188,A -85,B 0,C 180,E1 -10020.656,E2 -10020.656} C_VEL
LIN {X 0,Y 417.521,Z 271.941,A -85,B 0,C 180,E1 -10023.743,E2 -10023.743} C_VEL
LIN {X 0,Y 417.665,Z 267.192,A -85,B 0,C 180,E1 -10027.283,E2 -10027.283} C_VEL
LIN {X 0,Y 417.82,Z 263.99,A -85,B 0,C 180,E1 -10029.73,E2 -10029.73} C_VEL
LIN {X 0,Y 417.988,Z 260.715,A -85,B 0,C 180,E1 -10032.287,E2 -10032.287} C_VEL
LIN {X 0,Y 418.216,Z 257.197,A -85,B 0,C 180,E1 -10035.108,E2 -10035.108} C_VEL
LIN {X 0,Y 418.31,Z 253.971,A -85,B 0,C 180,E1 -10037.778,E2 -10037.778} C_VEL
LIN {X 0,Y 418.295,Z 252.412,A -85,B 0,C 180,E1 -10039.117,E2 -10039.117} C_VEL
LIN {X 0,Y 418.218,Z 251.399,A -85,B 0,C 180,E1 -10040.316,E2 -10040.316} C_VEL
LIN {X 0,Y 418.236,Z 251.39,A -85,B 0,C 180,E1 -10043.762,E2 -10043.762} C_VEL
LIN {X 0,Y 418.245,Z 251.391,A -85,B 0,C 180,E1 -10047.157,E2 -10047.157} C_VEL
LIN {X 0,Y 418.262,Z 251.385,A -85,B 0,C 180,E1 -10050.839,E2 -10050.839} C_VEL
LIN {X 0,Y 418.259,Z 251.385,A -85,B 0,C 180,E1 -10054.097,E2 -10054.097} C_VEL
LIN {X 0,Y 418.264,Z 251.383,A -85,B 0,C 180,E1 -10057.538,E2 -10057.538} C_VEL
LIN {X 0,Y 418.306,Z 251.378,A -85,B 0,C 180,E1 -10060.367,E2 -10060.367} C_VEL
LIN {X 0,Y 418.314,Z 251.377,A -85,B 0,C 180,E1 -10063.406,E2 -10063.406} C_VEL
LIN {X 0,Y 418.335,Z 251.378,A -85,B 0,C 180,E1 -10067,E2 -10067} C_VEL
LIN {X 0,Y 418.331,Z 251.377,A -85,B 0,C 180,E1 -10070.33,E2 -10070.33} C_VEL
LIN {X 0,Y 418.479,Z 251.358,A -85,B 0,C 180,E1 -10073.25,E2 -10073.25} C_VEL
LIN {X 0,Y 418.33,Z 251.375,A -85,B 0,C 180,E1 -10075.183,E2 -10075.183} C_VEL
LIN {X 0,Y 418.536,Z 251.35,A -85,B 0,C 180,E1 -10078.077,E2 -10078.077} C_VEL
LIN {X 0,Y 418.659,Z 251.334,A -85,B 0,C 180,E1 -10080.001,E2 -10080.001} C_VEL
LIN {X 0,Y 418.503,Z 251.354,A -85,B 0,C 180,E1 -10082.889,E2 -10082.889} C_VEL
LIN {X 0,Y 418.482,Z 251.359,A -85,B 0,C 180,E1 -10086.752,E2 -10086.752} C_VEL
LIN {X 0,Y 418.392,Z 251.368,A -85,B 0,C 180,E1 -10088.696,E2 -10088.696} C_VEL
LIN {X 0,Y 418.309,Z 251.378,A -85,B 0,C 180,E1 -10091.632,E2 -10091.632} C_VEL
LIN {X 0,Y 418.295,Z 251.382,A -85,B 0,C 180,E1 -10094.598,E2 -10094.598} C_VEL
LIN {X 0,Y 418.281,Z 251.385,A -85,B 0,C 180,E1 -10097.605,E2 -10097.605} C_VEL
LIN {X 0,Y 418.243,Z 251.389,A -85,B 0,C 180,E1 -10100.664,E2 -10100.664} C_VEL
LIN {X 0,Y 418.281,Z 251.386,A -85,B 0,C 180,E1 -10103.783,E2 -10103.783} C_VEL
LIN {X 0,Y 418.261,Z 251.388,A -85,B 0,C 180,E1 -10107.06,E2 -10107.06} C_VEL
LIN {X 0,Y 418.238,Z 251.391,A -85,B 0,C 180,E1 -10110.274,E2 -10110.274} C_VEL
LIN {X 0,Y 418.245,Z 251.389,A -85,B 0,C 180,E1 -10113.678,E2 -10113.678} C_VEL
LIN {X 0,Y 418.237,Z 251.388,A -85,B 0,C 180,E1 -10117.226,E2 -10117.226} C_VEL
LIN {X 0,Y 418.248,Z 251.387,A -85,B 0,C 180,E1 -10119.683,E2 -10119.683} C_VEL
LIN {X 0,Y 418.227,Z 251.388,A -85,B 0,C 180,E1 -10122.322,E2 -10122.322} C_VEL
LIN {X 0,Y 418.234,Z 251.382,A -85,B 0,C 180,E1 -10125.11,E2 -10125.11} C_VEL
LIN {X 0,Y 418.245,Z 251.557,A -85,B 0,C 180,E1 -10128.093,E2 -10128.093} C_VEL
LIN {X 0,Y 419.186,Z 257.016,A -85,B 0,C 180,E1 -10131.661,E2 -10131.661} C_VEL
LIN {X 0,Y 419.584,Z 261.076,A -85,B 0,C 180,E1 -10134.11,E2 -10134.11} C_VEL
LIN {X 0,Y 419.5,Z 265.195,A -85,B 0,C 180,E1 -10136.438,E2 -10136.438} C_VEL
LIN {X 0,Y 418.982,Z 271.406,A -85,B 0,C 180,E1 -10139.788,E2 -10139.788} C_VEL
LIN {X 0,Y 418.385,Z 278.751,A -85,B 0,C 180,E1 -10143.568,E2 -10143.568} C_VEL
LIN {X 0,Y 418.063,Z 285.117,A -85,B 0,C 180,E1 -10146.731,E2 -10146.731} C_VEL
LIN {X 0,Y 417.729,Z 291.496,A -85,B 0,C 180,E1 -10149.825,E2 -10149.825} C_VEL
LIN {X 0,Y 417.568,Z 296.921,A -85,B 0,C 180,E1 -10152.398,E2 -10152.398} C_VEL
LIN {X 0,Y 420.302,Z 310.403,A -85,B 0,C 180,E1 -10152.948,E2 -10152.948} C_VEL
LIN {X 0,Y 421.962,Z 322.89,A -85,B 0,C 180,E1 -10153.615,E2 -10153.615} C_VEL
LIN {X 0,Y 422.026,Z 328.163,A -85,B 0,C 180,E1 -10153.928,E2 -10153.928} C_VEL
LIN {X 0,Y 421.176,Z 340.316,A -85,B 0,C 180,E1 -10154.763,E2 -10154.763} C_VEL
LIN {X 0,Y 420.344,Z 350.947,A -85,B 0,C 180,E1 -10155.698,E2 -10155.698} C_VEL
LIN {X 0,Y 419.7,Z 360.071,A -85,B 0,C 180,E1 -10156.689,E2 -10156.689} C_VEL
LIN {X 0,Y 419.05,Z 369.207,A -85,B 0,C 180,E1 -10157.899,E2 -10157.899} C_VEL
LIN {X 0,Y 418.238,Z 378.123,A -85,B 0,C 180,E1 -10159.348,E2 -10159.348} C_VEL
LIN {X 0,Y 417.765,Z 385.317,A -85,B 0,C 180,E1 -10160.804,E2 -10160.804} C_VEL
LIN {X 0,Y 417.4,Z 391.077,A -85,B 0,C 180,E1 -10162.259,E2 -10162.259} C_VEL
LIN {X 0,Y 417.144,Z 395.692,A -85,B 0,C 180,E1 -10163.739,E2 -10163.739} C_VEL
LIN {X 0,Y 417.108,Z 399.092,A -85,B 0,C 180,E1 -10165.167,E2 -10165.167} C_VEL
LIN {X 0,Y 417.028,Z 402.158,A -85,B 0,C 180,E1 -10167.102,E2 -10167.102} C_VEL
LIN {X 0,Y 417.057,Z 403.097,A -85,B 0,C 180,E1 -10168.069,E2 -10168.069} C_VEL
LIN {X 0,Y 417.012,Z 403.639,A -85,B 0,C 180,E1 -10169.034,E2 -10169.034} C_VEL
LIN {X 0,Y 417.005,Z 403.748,A -85,B 0,C 180,E1 -10170,E2 -10170} C_VEL
LIN {X 0,Y 417.058,Z 402.803,A -85,B 0,C 180,E1 -10171.931,E2 -10171.931} C_VEL
LIN {X 0,Y 417.031,Z 401.741,A -85,B 0,C 180,E1 -10172.898,E2 -10172.898} C_VEL
LIN {X 0,Y 417.015,Z 400.223,A -85,B 0,C 180,E1 -10173.865,E2 -10173.865} C_VEL
LIN {X 0,Y 417.123,Z 397.158,A -85,B 0,C 180,E1 -10175.317,E2 -10175.317} C_VEL
LIN {X 0,Y 417.235,Z 393.023,A -85,B 0,C 180,E1 -10176.771,E2 -10176.771} C_VEL
LIN {X 0,Y 417.508,Z 386.69,A -85,B 0,C 180,E1 -10178.47,E2 -10178.47} C_VEL
LIN {X 0,Y 417.912,Z 379.788,A -85,B 0,C 180,E1 -10179.926,E2 -10179.926} C_VEL
LIN {X 0,Y 418.316,Z 372.732,A -85,B 0,C 180,E1 -10181.14,E2 -10181.14} C_VEL
LIN {X 0,Y 418.946,Z 364.231,A -85,B 0,C 180,E1 -10182.35,E2 -10182.35} C_VEL
LIN {X 0,Y 419.602,Z 353.705,A -85,B 0,C 180,E1 -10183.561,E2 -10183.561} C_VEL
LIN {X 0,Y 420.317,Z 341.847,A -85,B 0,C 180,E1 -10184.649,E2 -10184.649} C_VEL
LIN {X 0,Y 421.071,Z 329.92,A -85,B 0,C 180,E1 -10185.489,E2 -10185.489} C_VEL
LIN {X 0,Y 421.147,Z 322.461,A -85,B 0,C 180,E1 -10185.919,E2 -10185.919} C_VEL
LIN {X 0,Y 419.361,Z 309.379,A -85,B 0,C 180,E1 -10186.563,E2 -10186.563} C_VEL
LIN {X 0,Y 417.418,Z 297.108,A -85,B 0,C 180,E1 -10187,E2 -10187} C_VEL
LIN {X 0,Y 417.662,Z 290.228,A -85,B 0,C 180,E1 -10190.179,E2 -10190.179} C_VEL
LIN {X 0,Y 417.887,Z 283.622,A -85,B 0,C 180,E1 -10193.279,E2 -10193.279} C_VEL
LIN {X 0,Y 418.238,Z 276.988,A -85,B 0,C 180,E1 -10196.442,E2 -10196.442} C_VEL
LIN {X 0,Y 418.606,Z 270.358,A -85,B 0,C 180,E1 -10199.687,E2 -10199.687} C_VEL
LIN {X 0,Y 419.007,Z 263.759,A -85,B 0,C 180,E1 -10203.001,E2 -10203.001} C_VEL
LIN {X 0,Y 419.267,Z 259.273,A -85,B 0,C 180,E1 -10205.33,E2 -10205.33} C_VEL
LIN {X 0,Y 418.998,Z 255.919,A -85,B 0,C 180,E1 -10207.144,E2 -10207.144} C_VEL
LIN {X 0,Y 418.272,Z 251.385,A -85,B 0,C 180,E1 -10209.835,E2 -10209.835} C_VEL
LIN {X 0,Y 418.196,Z 251.391,A -85,B 0,C 180,E1 -10213.552,E2 -10213.552} C_VEL
LIN {X 0,Y 418.175,Z 251.395,A -85,B 0,C 180,E1 -10216.443,E2 -10216.443} C_VEL
LIN {X 0,Y 418.204,Z 251.391,A -85,B 0,C 180,E1 -10219.132,E2 -10219.132} C_VEL
LIN {X 0,Y 418.229,Z 251.39,A -85,B 0,C 180,E1 -10222.774,E2 -10222.774} C_VEL
LIN {X 0,Y 418.228,Z 251.39,A -85,B 0,C 180,E1 -10226.32,E2 -10226.32} C_VEL
LIN {X 0,Y 418.237,Z 251.386,A -85,B 0,C 180,E1 -10229.726,E2 -10229.726} C_VEL
LIN {X 0,Y 418.213,Z 251.39,A -85,B 0,C 180,E1 -10233.016,E2 -10233.016} C_VEL
LIN {X 0,Y 418.268,Z 251.386,A -85,B 0,C 180,E1 -10236.217,E2 -10236.217} C_VEL
LIN {X 0,Y 418.244,Z 251.386,A -85,B 0,C 180,E1 -10239.336,E2 -10239.336} C_VEL
LIN {X 0,Y 418.279,Z 251.383,A -85,B 0,C 180,E1 -10242.395,E2 -10242.395} C_VEL
LIN {X 0,Y 418.295,Z 251.379,A -85,B 0,C 180,E1 -10245.402,E2 -10245.402} C_VEL
LIN {X 0,Y 418.308,Z 251.379,A -85,B 0,C 180,E1 -10248.368,E2 -10248.368} C_VEL
LIN {X 0,Y 418.477,Z 251.358,A -85,B 0,C 180,E1 -10252.278,E2 -10252.278} C_VEL
LIN {X 0,Y 418.504,Z 251.355,A -85,B 0,C 180,E1 -10254.216,E2 -10254.216} C_VEL
LIN {X 0,Y 418.536,Z 251.351,A -85,B 0,C 180,E1 -10258.074,E2 -10258.074} C_VEL
LIN {X 0,Y 418.665,Z 251.335,A -85,B 0,C 180,E1 -10259.999,E2 -10259.999} C_VEL
LIN {X 0,Y 418.503,Z 251.354,A -85,B 0,C 180,E1 -10262.887,E2 -10262.887} C_VEL
LIN {X 0,Y 418.485,Z 251.356,A -85,B 0,C 180,E1 -10266.75,E2 -10266.75} C_VEL
LIN {X 0,Y 418.333,Z 251.376,A -85,B 0,C 180,E1 -10269.67,E2 -10269.67} C_VEL
LIN {X 0,Y 418.336,Z 251.375,A -85,B 0,C 180,E1 -10273,E2 -10273} C_VEL
LIN {X 0,Y 418.302,Z 251.378,A -85,B 0,C 180,E1 -10276.734,E2 -10276.734} C_VEL
LIN {X 0,Y 418.26,Z 251.386,A -85,B 0,C 180,E1 -10279.789,E2 -10279.789} C_VEL
LIN {X 0,Y 418.227,Z 251.388,A -85,B 0,C 180,E1 -10282.735,E2 -10282.735} C_VEL
LIN {X 0,Y 418.26,Z 251.384,A -85,B 0,C 180,E1 -10285.903,E2 -10285.903} C_VEL
LIN {X 0,Y 418.263,Z 251.386,A -85,B 0,C 180,E1 -10289.16,E2 -10289.16} C_VEL
LIN {X 0,Y 418.246,Z 251.386,A -85,B 0,C 180,E1 -10292.843,E2 -10292.843} C_VEL
LIN {X 0,Y 418.237,Z 251.385,A -85,B 0,C 180,E1 -10296.238,E2 -10296.238} C_VEL
LIN {X 0,Y 418.254,Z 251.383,A -85,B 0,C 180,E1 -10299.68,E2 -10299.68} C_VEL
LIN {X 0,Y 418.273,Z 251.381,A -85,B 0,C 180,E1 -10302.329,E2 -10302.329} C_VEL
LIN {X 0,Y 418.243,Z 251.387,A -85,B 0,C 180,E1 -10305.111,E2 -10305.111} C_VEL
LIN {X 0,Y 418.23,Z 251.385,A -85,B 0,C 180,E1 -10307.767,E2 -10307.767} C_VEL
LIN {X 0,Y 418.244,Z 251.389,A -85,B 0,C 180,E1 -10310.618,E2 -10310.618} C_VEL
LIN {X 0,Y 418.233,Z 251.386,A -85,B 0,C 180,E1 -10313.976,E2 -10313.976} C_VEL
LIN {X 0,Y 418.245,Z 251.385,A -85,B 0,C 180,E1 -10317.156,E2 -10317.156} C_VEL
LIN {X 0,Y 418.256,Z 251.384,A -85,B 0,C 180,E1 -10320.895,E2 -10320.895} C_VEL
LIN {X 0,Y 418.247,Z 251.388,A -85,B 0,C 180,E1 -10324.095,E2 -10324.095} C_VEL
LIN {X 0,Y 418.122,Z 251.4,A -85,B 0,C 180,E1 -10327.258,E2 -10327.258} C_VEL
LIN {X 0,Y 418.013,Z 251.454,A -85,B 0,C 180,E1 -10328.292,E2 -10328.292} C_VEL
LIN {X 0,Y 417.974,Z 255.49,A -85,B 0,C 180,E1 -10331.369,E2 -10331.369} C_VEL
LIN {X 0,Y 417.836,Z 259.552,A -85,B 0,C 180,E1 -10334.388,E2 -10334.388} C_VEL
LIN {X 0,Y 417.811,Z 263.613,A -85,B 0,C 180,E1 -10337.369,E2 -10337.369} C_VEL
LIN {X 0,Y 417.607,Z 269.101,A -85,B 0,C 180,E1 -10341.288,E2 -10341.288} C_VEL
LIN {X 0,Y 417.636,Z 271.868,A -85,B 0,C 180,E1 -10343.235,E2 -10343.235} C_VEL
LIN {X 0,Y 417.518,Z 276.088,A -85,B 0,C 180,E1 -10346.109,E2 -10346.109} C_VEL
LIN {X 0,Y 419.885,Z 289.119,A -85,B 0,C 180,E1 -10346.612,E2 -10346.612} C_VEL
LIN {X 0,Y 421.733,Z 299.079,A -85,B 0,C 180,E1 -10347.134,E2 -10347.134} C_VEL
LIN {X 0,Y 421.12,Z 311.074,A -85,B 0,C 180,E1 -10347.848,E2 -10347.848} C_VEL
LIN {X 0,Y 420.48,Z 321.933,A -85,B 0,C 180,E1 -10348.683,E2 -10348.683} C_VEL
LIN {X 0,Y 419.832,Z 333.01,A -85,B 0,C 180,E1 -10349.76,E2 -10349.76} C_VEL
LIN {X 0,Y 419.109,Z 342.884,A -85,B 0,C 180,E1 -10350.961,E2 -10350.961} C_VEL
LIN {X 0,Y 418.411,Z 352.463,A -85,B 0,C 180,E1 -10352.407,E2 -10352.407} C_VEL
LIN {X 0,Y 417.944,Z 360.082,A -85,B 0,C 180,E1 -10353.857,E2 -10353.857} C_VEL
LIN {X 0,Y 417.545,Z 366.221,A -85,B 0,C 180,E1 -10355.312,E2 -10355.312} C_VEL
LIN {X 0,Y 417.455,Z 369.368,A -85,B 0,C 180,E1 -10356.211,E2 -10356.211} C_VEL
LIN {X 0,Y 416.661,Z 371.696,A -85,B 0,C 180,E1 -10356.949,E2 -10356.949} C_VEL
LIN {X 0,Y 413.588,Z 374.927,A -85,B 0,C 180,E1 -10358.173,E2 -10358.173} C_VEL
LIN {X 0,Y 411.042,Z 376.965,A -85,B 0,C 180,E1 -10359.186,E2 -10359.186} C_VEL
LIN {X 0,Y 409.956,Z 378.235,A -85,B 0,C 180,E1 -10359.983,E2 -10359.983} C_VEL
LIN {X 0,Y 409.869,Z 378.544,A -85,B 0,C 180,E1 -10360.255,E2 -10360.255} C_VEL
LIN {X 0,Y 409.901,Z 380.076,A -85,B 0,C 180,E1 -10361.873,E2 -10361.873} C_VEL
LIN {X 0,Y 409.804,Z 380.45,A -85,B 0,C 180,E1 -10362.882,E2 -10362.882} C_VEL
LIN {X 0,Y 409.783,Z 380.426,A -85,B 0,C 180,E1 -10363.893,E2 -10363.893} C_VEL
LIN {X 0,Y 409.813,Z 379.993,A -85,B 0,C 180,E1 -10364.906,E2 -10364.906} C_VEL
LIN {X 0,Y 409.954,Z 378.714,A -85,B 0,C 180,E1 -10366.26,E2 -10366.26} C_VEL
LIN {X 0,Y 410.113,Z 376.048,A -85,B 0,C 180,E1 -10367.966,E2 -10367.966} C_VEL
LIN {X 0,Y 410.39,Z 372.155,A -85,B 0,C 180,E1 -10369.635,E2 -10369.635} C_VEL
LIN {X 0,Y 410.732,Z 367.761,A -85,B 0,C 180,E1 -10371.058,E2 -10371.058} C_VEL
LIN {X 0,Y 411.258,Z 361.418,A -85,B 0,C 180,E1 -10372.664,E2 -10372.664} C_VEL
LIN {X 0,Y 411.915,Z 353.932,A -85,B 0,C 180,E1 -10374.172,E2 -10374.172} C_VEL
LIN {X 0,Y 412.625,Z 345.883,A -85,B 0,C 180,E1 -10375.486,E2 -10375.486} C_VEL
LIN {X 0,Y 413.432,Z 336.15,A -85,B 0,C 180,E1 -10376.774,E2 -10376.774} C_VEL
LIN {X 0,Y 414.314,Z 325.615,A -85,B 0,C 180,E1 -10377.891,E2 -10377.891} C_VEL
LIN {X 0,Y 415.093,Z 314.31,A -85,B 0,C 180,E1 -10378.85,E2 -10378.85} C_VEL
LIN {X 0,Y 415.888,Z 303.346,A -85,B 0,C 180,E1 -10379.568,E2 -10379.568} C_VEL
LIN {X 0,Y 415.728,Z 299.33,A -85,B 0,C 180,E1 -10379.806,E2 -10379.806} C_VEL
LIN {X 0,Y 413.378,Z 287.985,A -85,B 0,C 180,E1 -10380.462,E2 -10380.462} C_VEL
LIN {X 0,Y 410.319,Z 276.435,A -85,B 0,C 180,E1 -10381.003,E2 -10381.003} C_VEL
LIN {X 0,Y 410.498,Z 271.834,A -85,B 0,C 180,E1 -10384.4,E2 -10384.4} C_VEL
LIN {X 0,Y 410.603,Z 268.657,A -85,B 0,C 180,E1 -10386.802,E2 -10386.802} C_VEL
LIN {X 0,Y 410.773,Z 264.969,A -85,B 0,C 180,E1 -10389.656,E2 -10389.656} C_VEL
LIN {X 0,Y 411,Z 260.582,A -85,B 0,C 180,E1 -10393.155,E2 -10393.155} C_VEL
LIN {X 0,Y 411.228,Z 257.267,A -85,B 0,C 180,E1 -10395.871,E2 -10395.871} C_VEL
LIN {X 0,Y 411.26,Z 253.901,A -85,B 0,C 180,E1 -10398.755,E2 -10398.755} C_VEL
LIN {X 0,Y 411.184,Z 252.275,A -85,B 0,C 180,E1 -10400.275,E2 -10400.275} C_VEL
LIN {X 0,Y 411.182,Z 252.268,A -85,B 0,C 180,E1 -10403.448,E2 -10403.448} C_VEL
LIN {X 0,Y 411.195,Z 252.269,A -85,B 0,C 180,E1 -10406.874,E2 -10406.874} C_VEL
LIN {X 0,Y 411.228,Z 252.262,A -85,B 0,C 180,E1 -10410.643,E2 -10410.643} C_VEL
LIN {X 0,Y 411.226,Z 252.263,A -85,B 0,C 180,E1 -10413.62,E2 -10413.62} C_VEL
LIN {X 0,Y 411.197,Z 252.262,A -85,B 0,C 180,E1 -10416.854,E2 -10416.854} C_VEL
LIN {X 0,Y 411.254,Z 252.256,A -85,B 0,C 180,E1 -10420.032,E2 -10420.032} C_VEL
LIN {X 0,Y 411.253,Z 252.257,A -85,B 0,C 180,E1 -10423.132,E2 -10423.132} C_VEL
LIN {X 0,Y 411.294,Z 252.255,A -85,B 0,C 180,E1 -10426.897,E2 -10426.897} C_VEL
LIN {X 0,Y 411.283,Z 252.256,A -85,B 0,C 180,E1 -10430.162,E2 -10430.162} C_VEL
LIN {X 0,Y 411.446,Z 252.234,A -85,B 0,C 180,E1 -10433.134,E2 -10433.134} C_VEL
LIN {X 0,Y 411.3,Z 252.251,A -85,B 0,C 180,E1 -10435.1,E2 -10435.1} C_VEL
LIN {X 0,Y 411.505,Z 252.226,A -85,B 0,C 180,E1 -10438.044,E2 -10438.044} C_VEL
LIN {X 0,Y 411.629,Z 252.21,A -85,B 0,C 180,E1 -10440.001,E2 -10440.001} C_VEL
LIN {X 0,Y 411.458,Z 252.232,A -85,B 0,C 180,E1 -10442.938,E2 -10442.938} C_VEL
